// TwinCAT 3 PLC project R1_TemplatePLC
// ProgramVersion: 3.1.4022.3
// libraries:
//   Tc2_Drive, * (Beckhoff Automation GmbH)
//   Tc2_EtherCAT, * (Beckhoff Automation GmbH)
//   Tc2_IoFunctions, * (Beckhoff Automation GmbH)
//   Tc2_MC2, * (Beckhoff Automation GmbH)
//   Tc2_MC2_Drive, * (Beckhoff Automation GmbH)
//   Tc2_MDP, * (Beckhoff Automation GmbH)
//   Tc2_Standard, * (Beckhoff Automation GmbH)
//   Tc2_SUPS, * (Beckhoff Automation GmbH)
//   Tc2_System, * (Beckhoff Automation GmbH)
//   Tc2_Utilities, * (Beckhoff Automation GmbH)
//   Tc3_EventLogger, * (Beckhoff Automation GmbH)
//   Tc3_Module, * (Beckhoff Automation GmbH)
//   VisuDialogs, * (System)
// project tree:
//   DUTs/DUTsAxisOnline/FBsIO/ ST_FBGetDriveRefIO.TcDUT (not stored), ST_FBHoldingBrakeCtrlIO.TcDUT (not stored), ST_FBMotorMonitoringIO.TcDUT (not stored), ST_FBNcSWLimitSwitchCtrlIO.TcDUT (not stored), ST_FBReadChannelErrorCodeIO.TcDUT (not stored), ST_FBSetPositionOffsetIO.TcDUT, ST_McAxisOnlineErrorCollection.TcDUT, ST_McAxisStatus.TcDUT (not stored), ST_MCHaltIO.TcDUT (not stored), ST_MCHomeIO.TcDUT (not stored), ST_MCJogIO.TcDUT (not stored), ST_MCMoveAbsoluteIO.TcDUT (not stored), ST_MCMoveModuloIO.TcDUT (not stored), ST_MCMoveRelativeIO.TcDUT (not stored), ST_MCMoveVelocityIO.TcDUT (not stored), ST_MCPowerIO.TcDUT (not stored), ST_MCReadDriveAddressIO.TcDUT (not stored), ST_MCReadParameterSetIO.TcDUT (not stored), ST_MCResetIO.TcDUT (not stored), ST_MCSetPositionIO.TcDUT (not stored), ST_MCStopIO.TcDUT (not stored)
//   DUTs/DUTsAxisOnline/ ST_AX5000Diag.TcDUT (not stored), ST_McAxisOnline.TcDUT (not stored)
//   DUTs/DUTsDiagnostics/ ST_FrmWcDiag.TcDUT, ST_KBusState.TcDUT
//   DUTs/DUTsOther/ E_MachineCommand.TcDUT (not stored), E_MachineMode.TcDUT, E_MachineState.TcDUT (not stored)
//   / GlobalTextList.TcGTLO, PlcTask.TcTTO, Visualization Manager.TcVMO (not stored)
//   GVLs/ GVL.TcGVL, GVL_EventLogger_Simple.TcGVL, GVL_IO.TcGVL, GVL_Machine.TcGVL
//   GVLs/GVLsDiagnostics/ GVL_Checks.TcGVL
//   POUs/ MAIN.TcPOU, P_ErrorCollection.TcPOU, P_EventLogger_Simple.TcPOU, P_Initialization.TcPOU, P_ModeStateManager.TcPOU, P_Template.TcPOU, P_Template_SAFETY.TcPOU
//   POUs/POUsAxisOnline/AX5000/ FB_AxisDiag.TcPOU, FB_ChangeEtherCATSlaveState.TcPOU, FB_HoldingBrakeCtrlAX5000.TcPOU (not stored), FB_McAxisOnlineAX5000.TcPOU, FB_MotorMonitoringAX5000.TcPOU, FB_SetPositionOffset.TcPOU, F_AX5xErrMsg.TcPOU
//   POUs/POUsAxisOnline/AX8000/ FB_HoldingBrakeCtrlAX8000.TcPOU, FB_McAxisOnlineAX8000.TcPOU, FB_MotorMonitoringAX8000.TcPOU, FB_ReadChannelErrorCodeAX8000.TcPOU, F_AX8xErrMsg.TcPOU
//   POUs/POUsAxisOnline/EL72xx/ FB_HoldingBrakeCtrlEL72xx.TcPOU, FB_McAxisOnlineEL72xx.TcPOU, FB_MotorMonitoringEL72xx.TcPOU, FB_ReadChannelErrorCodeEL72xx.TcPOU, F_EL72ErrMsg.TcPOU
//   POUs/POUsAxisOnline/FBs/ FB_FilterEx.TcPOU (not stored), FB_GetDriveRef.TcPOU (not stored), FB_NcSWLimitSwitchCtrl.TcPOU (not stored), F_AxErrMsg.TcPOU
//   POUs/POUsAxisOnline/NC/ FB_McAxisOnlineNC.TcPOU
//   POUs/POUsDiagnostics/Checks/ CheckBounds.TcPOU, CheckDivDInt.TcPOU, CheckDivLInt.TcPOU, CheckDivLReal.TcPOU, CheckDivReal.TcPOU, CheckPointer.TcPOU, CheckRangeSigned.TcPOU, CheckRangeUnsigned.TcPOU
//   POUs/POUsDiagnostics/FB/ FB_AntiBlinkAlarmFilter.TcPOU, FB_TaskInfo.TcPOU (not stored)
//   POUs/POUsDiagnostics/ P_Checks.TcPOU, P_EtherCAT_ChangeCounter.TcPOU, P_EtherCAT_Diag.TcPOU, P_KBus.TcPOU, P_Persistent.TcPOU, P_SystemDiagnostics.TcPOU, P_SystemDiag_EventLog.TcPOU, P_SystemInfo.TcPOU, P_TaskInfo.TcPOU (not stored)
//   POUs/POUsOther/ FB_AutostartPLCHMI.TcPOU, FB_Blink_S.TcPOU
//   VISUs/VISUsAxisOnline/ PH_AxisOnline.TcVIS, PH_MotorMonitoring.TcVIS, PH_NcAxis.TcVIS
//   VISUs/ VIS_SM.TcVIS
// real-time tasks:
//   TASK PlcTask: cycle T#10ms, priority 20, ADS port 350
//   TASK SafetyTask: cycle T#10ms, priority 21, ADS port 351

CONFIGURATION R1_TemplatePLC
    RESOURCE PLC ON TwinCAT3
        TASK PlcTask(INTERVAL := T#10ms, PRIORITY := 20);
        PROGRAM MAIN WITH PlcTask : MAIN;
    END_RESOURCE
END_CONFIGURATION

// ---- DUTs/DUTsAxisOnline/FBsIO/ST_FBSetPositionOffsetIO.TcDUT
//==================================================================================================
//							Beckhoff Automation Poland
//									23.05.2018
//	Struktura zawierajaca I/O odpowiedniego bloku
//  v1.1	|| TC v 3.1.4022.16		|| - zmiana nazwy struktury usuniete CoE
//  v1.0	|| TC v 3.1.4022.16		|| - pierwsza wersja
//==================================================================================================
TYPE ST_FBSetPositionOffsetIO:
STRUCT
	bExecute						: BOOL;								// Rising edge executes cmd
	lrPosition						: LREAL;
	bRelative						: BOOL;
	eFeedback						: Tc2_MC2_Drive.E_PositionOffsetFeedback;
	eMemory							: Tc2_MC2_Drive.E_PositionOffsetMemory;
	bBusy							: BOOL;
	bError							: BOOL;
	udiErrorID						: UDINT;
	uiSecErrId						: UINT;								// Sercos Error ID for AX5000, CanOpen error ID for AX8000
END_STRUCT
END_TYPE

// ---- DUTs/DUTsAxisOnline/FBsIO/ST_McAxisOnlineErrorCollection.TcDUT
//==================================================================================================
//							Beckhoff Automation Poland
//									7.12.2018
//	Struktura zawierajaca wszsytkie bbledy AxisOnline
//  v1.1	|| TC v 3.1.4022.27		|| - dodane opisy bledow w formie zmiennych typu string
//  v1.0	|| TC v 3.1.4022.16		|| - pierwsza wersja
//==================================================================================================
TYPE ST_McAxisOnlineErrorCollection :
STRUCT
	// Error Collection
	bError							: BOOL;						// General Error flag - all error, FB, NC, drive, communication...
	bNcError						: BOOL;
	bFBError						: BOOL;						// Mc FB error
	bCommunicationError				: BOOL;						// ADS, CoE (AX8000), SoE (AX5000)...
	bDriveError						: BOOL;
	uiAdsErrorID					: UINT;						// Forwarded output FB_CoERead_ByDriveRef
	uiSecErrorID					: UINT;						// Sercos Error ID for AX5000, CanOpen error ID for AX8000
	udiErrorID						: UDINT;					// Set Position Offset FB error ID
	udiNcErrorID					: UDINT;					// Nc ErrorID
	{attribute 'displaymode':='hex'}
	udiNcErrorIDHex					: UDINT;					// Nc ErrorID
	udiFBErrorID					: UDINT;					// FB ErrorID
	{attribute 'displaymode':='hex'}
	udiFBErrorIDHex					: UDINT;					// FB ErrorID

	uiDriveErrorID					: UINT;						// 603F Error code	0x603F (Ch A)/ 0x683F (Ch B) 	UINT16
	{attribute 'displaymode':='hex'}
	uiDriveErrorIDHex				: UINT;						// 603F Error code	0x603F (Ch A)/ 0x683F (Ch B) 	UINT16
	sNcError						: STRING(255);				// Error description
	sDriveError						: STRING(255);				// Error description
END_STRUCT
END_TYPE

// ---- DUTs/DUTsDiagnostics/ST_FrmWcDiag.TcDUT
TYPE ST_FrmWcDiag :
STRUCT
	iNum					:DINT;
	sBin					:String;
END_STRUCT
END_TYPE

// ---- DUTs/DUTsDiagnostics/ST_KBusState.TcDUT
TYPE ST_KBusState :							// K_Bus_diagnostic flags structure
STRUCT
		bK_BusErr				:	BOOL;	// Bit 0 = K-Bus Err
		bTerminalStateErr		:	BOOL;	// Bit 1 = Terminal State Err
		bProcessDataLengthErr	:	BOOL;	// Bit 2 = Process Data Length Err
		bK_BusInvalid			:	BOOL;	// Bit 7 = K-Bus invalid
		bNoValidInputs			:	BOOL;	// Bit 8 = No valid Inputs
		bK_BusInputUpdateBusy	:	BOOL;	// Bit 9 = K-Bus Input Update busy
		bK_BusOutputUpdateBusy	:	BOOL;	// Bit 10 = K-Bus Output Update busy
		bWatchDogErr			:	BOOL;	// Bit 11 = Watchdog Err
		bAcycFunctionActive		:	BOOL;	// Bit 15 = Acyc. Function atcive (e.g. K-Bus Reset)
END_STRUCT
END_TYPE

// ---- DUTs/DUTsOther/E_MachineMode.TcDUT
//==================================================================================================
//							Beckhoff Automation Poland
//									22.12.2016
//	Typ glownej tablicy zdarzen historycznych
// 	v1.1	|| TC v 3.1.4022.25		|| - zamiana nazwy trybu poczatkowego na eInitialization
// 	v1.0	|| TC v 3.1.4020.28		|| - pierwsza wersja
//==================================================================================================
{attribute 'strict'}
{attribute 'qualified_only'}
TYPE E_MachineMode :
(
	eInitialization			:= 0,
	eManual					:= 1,
	eMaintenance			:= 2,
	eAutomatic				:= 3,
	eSemiAutomatic			:= 4,
	eFirstFilling			:= 5,
	eEmptying				:= 6
);
END_TYPE

// ---- GVLs/GVL.TcGVL
{attribute 'qualified_only'}
VAR_GLOBAL CONSTANT
	byNoOfAxes 							: BYTE:= 10; 			// Liczba osi
END_VAR
VAR_GLOBAL
	Axis								: ARRAY [1..byNoOfAxes] OF AXIS_REF;
	stMcAxisOnline						: ARRAY [1..byNoOfAxes] OF ST_McAxisOnline;
	//
	bAllUnitsReady						: BOOL;					// All machine units are OK, and ready to operate
	bGeneralOK							: BOOL;					// There is no Warning, Error or Fatal Error - just when it's true - You can operate
	bGeneralWarning						: BOOL;					// Warning - just message/event - no reaction
	bGeneralError						: BOOL;					// Error - machine has to stop, start is possible from this position
	bGeneralFatalError					: BOOL;					// Fatal error causes machine stop. You have to go back for cycle begin.

	// 
	bRestartRequired					: BOOL;					// In case of fatal error, when whole process restart required
	bMuteGeneralError					: BOOL;					// Just for service/maitenance - if You are aware of consequences You can force muting mode
	bMuteGeneralFatalError				: BOOL;					// Just for service/maitenance - if You are aware of consequences You can force muting mode
END_VAR

// ---- GVLs/GVLsDiagnostics/GVL_Checks.TcGVL
{attribute 'qualified_only'}
VAR_GLOBAL PERSISTENT
	dCheckBounds					: DINT;			// Licznik przekroczen zakresu indexow, np. tablic
	dCheckDivDInt					: DINT;			// Licznik prob dzielenia Dint przez 0
	dCheckDivLInt					: DINT; 		// Licznik prob dzielenia LInt przez 0
	dCheckDivLReal					: DINT; 		// Licznik prob dzielenia LREAL przez 0
	dCheckDivReal					: DINT; 		// Licznik prob dzielenia REAL przez 0
	dCheckRangeSigned				: DINT;			// Licznik przekroczen liczby znakowej
	dCheckRangeUnsigned				: DINT; 		// Licznik przekroczen liczby bezznakowej
END_VAR

// ---- GVLs/GVL_EventLogger_Simple.TcGVL
{attribute 'qualified_only'}
VAR_GLOBAL
	arrMessageTriggers		: ARRAY [1..nMaxNumMessages] OF BOOL; // auto clear
	arrWarningTriggers		: ARRAY [1..nMaxNumWarnings] OF BOOL; // auto clear
	arrErrorTriggers 		: ARRAY [1..nMaxNumErrors] OF BOOL; // manual clear
	arrErrorConfirmations	: ARRAY [1..nMaxNumErrors] OF BOOL; // auto clear
END_VAR
VAR_GLOBAL CONSTANT
	nMaxNumMessages 	: UDINT := 3;
	nMaxNumWarnings 	: UDINT := 3;
	nMaxNumErrors 		: UDINT := 3;
END_VAR

// ---- GVLs/GVL_IO.TcGVL
{attribute 'qualified_only'}
VAR_GLOBAL
// =============== SAMPLE NAMES =================

	di_PBStart 					AT %I*	: BOOL;					// Push button - Start
	di_PBStop 					AT %I*	: BOOL;					// Push button - Stop
	di_PBReset 					AT %I*	: BOOL;					// Push button - Reset
// ==============================================
// =================== SAFETY ===================
	bSAFETY_Error				AT %I*	: BOOL;
	bSAFETY_ResetCMD 			AT %Q*	: BOOL;
	bSAFETY_ResetBusy			AT %I*	: BOOL;
	bSAFETY_PermissionSS1		AT %I*	: BOOL; 				// Sygnal NC - TRUE - pozwolenie na prace
	bSAFETY_PermissionSS2		AT %I*	: BOOL; 				// Sygnal NC - TRUE - pozwolenie na prace
// ======== Error and states collection =========
	dwGroupErrors				AT %I*	: DWORD;				// Group Error collection - Communication, FB, Other...
	dwAXStatesSTO				AT %I*	: DWORD;
	dwAXStatesSOS				AT %I*	: DWORD;
	dwAXErrors					AT %I*	: DWORD;
END_VAR

// ---- GVLs/GVL_Machine.TcGVL
{attribute 'qualified_only'}
VAR_GLOBAL
	eMode									: E_MachineMode := E_MachineMode.eInitialization;	// Global machine mode
																						(*	eInitialization			:= 0,
																							eManual					:= 1,
																							eMaintenance			:= 2,
																							eAutomatic				:= 3,
																							eSemiAutomatic			:= 4,
																							eFirstFilling			:= 5,
																							eEmptying				:= 6	*)
																							
	eCommand								: E_MachineCommand; 							// Global machine command
																						(*	eAbort	  				:= 10,
																							eStop	  				:= 20,
																							eRun 	  				:= 30,
																							eReset	  				:= 40	*)
																							
	eState									: E_MachineState; 								// Global machine state
																						(*	eIdle					:= 0,
																							eAborting				:= 10,
																							eAborted				:= 20,
																							eStopping				:= 30,
																							eStopped				:= 40,
																							eStarting				:= 50,
																							eRunning				:= 60,
																							eReseting				:= 70,
																							eError					:= 1000	*)
END_VAR

// ---- POUs/MAIN.TcPOU
//==================================================================================================
//							Beckhoff Automation Poland
//									02.11.2018
//	Projekt startowy
// 	v1.2	|| TC v 3.1.4022.4		|| - zmiana wywolania osi
// 	v1.1	|| TC v 3.1.4020.32		|| - Aktualizacja
// 	v1.0	|| TC v 3.1.4020.28		|| - Pierwsza wersja
//==================================================================================================
PROGRAM MAIN
VAR
END_VAR

P_SystemDiagnostics();

P_EventLogger_Simple();

P_ErrorCollection();

P_ModeStateManager();

P_Template_SAFETY(eMachineMode:= GVL_Machine.eMode, eMachineCommand:= GVL_Machine.eCommand, eMachineState=> , bError=> );

P_Template(eMachineMode:= GVL_Machine.eMode, eMachineCommand:= GVL_Machine.eCommand, eMachineState=> , Axis1 := GVL.Axis[1]);
(*
P_Template_CAM(	eMachineMode		:= GVL_Machine.eMode, 
				eMachineCommand		:= GVL_Machine.eCommand, 
				eMachineState		=> GVL_Machine.eState,
				Axis1				:= GVL.Axis[1], 
				Axis2				:= GVL.Axis[2], 
				Axis3				:= GVL.Axis[3]);
*)

END_PROGRAM

// ---- POUs/POUsDiagnostics/P_SystemDiagnostics.TcPOU
//==================================================================================================
//							Beckhoff Automation Poland
//									2.11.2018
//					Program zbiorczy diagnostyki systemu
// 
//	v1.4 	|| TC v 3.1.4022.25 	|| Dodany state machine
//	v1.3 	|| TC v 3.1.4022.20 	|| Usuniete P_MDP, dodany podprogram EventLoggera P_SystemDiag_EventLog
//	v1.2 	|| TC v 3.1.4020.32 	|| Dodane P_EtherCAT_ChangeCounter
//	v1.1 	|| TC v 3.1.4020.14 	|| Dodane wyjscia bOk, bWarning, bError
//	v1.0 	|| TC v 3.1.4020.0 		|| Pierwsza wersja
//==================================================================================================
PROGRAM P_SystemDiagnostics
VAR_INPUT
	eMachineMode							: E_MachineMode; 		// Machine mode
	eMachineCommand							: E_MachineCommand; 	// Command from top level state program
END_VAR
VAR_OUTPUT
	eMachineState							: E_MachineState;
	bOK										: BOOL;					// Brak bledow i ostrzezen
	bWarning								: BOOL;					// Ostrzezenie
	bError									: BOOL;					// Zbiorcza flaga bledow
END_VAR
VAR
END_VAR

P_SystemInfo(bConfirm:=);
P_Persistent();
P_EtherCAT_Diag();
P_EtherCAT_ChangeCounter(bReset := );
P_KBus();
P_Checks(bReset := );
P_TaskInfo();

// Machine mode change over
CASE eMachineMode OF
	
	E_MachineMode.eInitialization:
		; // Do nothing
	
ELSE
	
	// Set flags
	bError										:= P_SystemInfo.bError OR P_Persistent.bError OR P_EtherCAT_Diag.bError OR P_EtherCAT_ChangeCounter.bError OR P_KBus.bError OR P_Checks.bError OR P_TaskInfo.bError;
	bWarning									:= P_SystemInfo.bWarning OR P_Persistent.bWarning OR P_EtherCAT_Diag.bWarning OR P_EtherCAT_ChangeCounter.bWarning OR P_KBus.bWarning OR P_Checks.bWarning OR P_TaskInfo.bWarning;
	bOk											:= NOT (bError OR bWarning);
	
	// State machine
	CASE eMachineState OF
	
		E_MachineState.eIdle, E_MachineState.eStopping, E_MachineState.eStopped, E_MachineState.eStarting, E_MachineState.eAborting, E_MachineState.eAborted:

			// Ignore global commands eAbort, eRun, eStop, eReset, eRestart
			// Set eRunning state
			eMachineState 						:= E_MachineState.eRunning;

		E_MachineState.eRunning:
		
			// Ignore global commands eAbort, eRun, eStop, eReset, eRestart
			// If error go to error state
			IF bError THEN
				eMachineState					:= E_MachineState.eError;
			END_IF
	
		E_MachineState.eRestarting, E_MachineState.eReseting:

			// Reset/Restart only if not OK
			P_EtherCAT_ChangeCounter.bReset		:= NOT P_EtherCAT_ChangeCounter.bOK;
			P_Checks.bReset						:= NOT P_Checks.bOK;
			IF NOT bError THEN
				eMachineState					:= E_MachineState.eRunning;
			END_IF

		E_MachineState.eError:
	
			IF eMachineCommand = E_MachineCommand.eReset THEN
				eMachineState					:= E_MachineState.eReseting;
			END_IF
	
			IF eMachineCommand = E_MachineCommand.eRestart THEN
				eMachineState					:= E_MachineState.eRestarting;
			END_IF
	
	END_CASE
	
END_CASE

// Log to events - You can switch it off in Initialization phase
P_SystemDiag_EventLog();

END_PROGRAM

// ---- POUs/POUsDiagnostics/P_SystemInfo.TcPOU
//==================================================================================================
//							Beckhoff Automation Poland
//									P_SystemInfo
//									31.10.2018
//					Program odczytujący informacje o TC Runtime
// 
//	v1.2 	|| TC v 3.1.4022.25 	|| - bOK dodane BSOD i sprawdzenie licencji
//	v1.1 	|| TC v 3.1.4020.14 	|| - Dodane wyjscia bOk, bWarning, bError
//	v1.0 	|| TC v 3.1.4020.0 		|| - Pierwsza wersja
//==================================================================================================
PROGRAM P_SystemInfo
VAR_INPUT
	bConfirm					: BOOL;					// Potwierdzenie bledu/ostrzezenia persistentow - blad/ostrzezenie nie znika, my usuwamy flage error lub warning
END_VAR
VAR_OUTPUT
	bOK							: BOOL;					// Zmienne wczytane prawidlowo
	bWarning					: BOOL;					// Zmienne wczytane z pliku zapasowego
	bError						: BOOL;					// Nie wczytano zmiennych
END_VAR
VAR
	sStartTime					: STRING;				// Przekonwertowany czas
END_VAR

//_AppInfo.ObjId; 			(* Object ID of the PLC project instance *)
//_AppInfo.TaskCnt;			(* The number of tasks in the actual runtime system *)
//_AppInfo.OnlineChangeCnt;	(* The number of online changes made since the last complete download. *)
//_AppInfo.Flags;				(* Reserved for future use *)
//_AppInfo.AdsPort; 			(* ADS port of PLC application *)
bOK							:= (_AppInfo.BootDataLoaded OR bConfirm) AND NOT _AppInfo.LicensesPending AND NOT _AppInfo.BSODOccured;	(* PERSISTENT variables: LOADED (without error) *)
bWarning					:= _AppInfo.OldBootData AND NOT bConfirm;	(* PERSISTENT variables: INVALID (the back-up copy was loaded, since no valid data was present) *)
bError						:= NOT bOK AND NOT bWarning;
//_AppInfo.KeepOutputsOnBP;	(* The flag can be set to avoid that the outputs are zero-filled if a breakpoint is reached. The task keeps running. Only the execution of PLC code is interrupted. *)
//_AppInfo.TComSrvPtr;		(* Pointer to TcCOM Object Server *)
//_AppInfo.AppName;			(* TwinCAT generated name containing the port number. *)
//_AppInfo.ProjectName;		(* The name of the PLC project. *)
sStartTime					:= DELETE(DT_TO_STRING(_AppInfo.AppTimestamp),3,1);(* Date and time of application start *)
(*_AppInfo.BSODOccured;
_AppInfo.LicensesPending;
_AppInfo.ShutdownInProgress;*)

END_PROGRAM

// ---- POUs/POUsDiagnostics/P_Persistent.TcPOU
//==================================================================================================
//							Beckhoff Automation Poland
//									25.04.2018
//		Program obslugujacy pamiec nieulotna 
// 	v1.3	|| TC v 3.1.4022.16		|| - Przeniesienie logowania do EvenLogger'a do programu P_SystemDiag_EventLog
// 	v1.2	|| TC v 3.1.4022.0		|| - Dodanie akcji UPS
//	v1.1 	|| TC v 3.1.4020.14 	|| - Dodane wyjscia bOk, bWarning, bError
//	v1.0 	|| TC v 3.1.4020.0 		|| - Pierwsza wersja
//==================================================================================================
PROGRAM P_Persistent
VAR_INPUT
	bWrite						: BOOL;						// Zapis na rozkaz - tylko dla iType = 0 lub nieokreslonego, gdy używany jest FB_WritePersistentData
	tInterval					: TIME := T#1H;				// Czestotliwosc zapisu na karte CF - tylko dla iType = 0 lub nieokreslonego, gdy używany jest FB_WritePersistentData
END_VAR
VAR_OUTPUT
	// Brak obslugi
	bOK							: BOOL := TRUE;				// Brak bledow i ostrzezen
	bWarning					: BOOL;						// Ostrzezenie
	bError						: BOOL;						// Zbiorcza flaga bledow
END_VAR
VAR
	iType						: INT := 0;					(* typ zapisu persistent:
																0: standardowo - na zadanie oraz co okreslony czas
																10: FB_S_UPS, np: CX50x0,C6915-0000,CP62xx-0020,CP77xx-0030
																20: FB_S_UPS_CB3011, np: CP66xx-0020, CP26xx-0000
																30: FB_S_UPS_CX51x0, np: CX51x0
																40: FB_S_UPS_CX9020_U900, np: CX9020 *)
	fbS_UPS						: FB_S_UPS;
	fbS_UPS_CB3011				: FB_S_UPS_CB3011;
	fbS_UPS_CX51x0				: FB_S_UPS_CX51x0;
	fbS_UPS_CX9020_U900			: FB_S_UPS_CX9020_U900;
	fbS_UPS_BAPI				: FB_S_UPS_BAPI;
	// Obsługa ogólna
	fbWritePersistentData 		: FB_WritePersistentData;	// Blok zapisu
	T1							: TON;						// Timer zapisu
END_VAR

CASE iType OF
	0:
		A_WritePersistentData();
		
	10:
	
		A_fbS_UPS();
		
	20:
		
		A_fbS_UPS_CB3011();
		
	30:
	
		A_fbS_UPS_CX51x0();
		
	40:
	
		A_fbS_UPS_CX9020_U900();
		
	50:
	
		A_fbS_UPS_BAPI();
		
ELSE
		A_WritePersistentData();		
		
END_CASE

ACTION A_fbS_UPS:
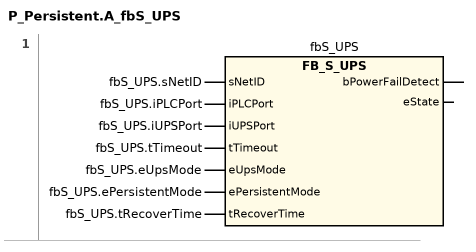
// NETWORK 1
fbS_UPS(
    sNetID := fbS_UPS.sNetID,
    iPLCPort := fbS_UPS.iPLCPort,
    iUPSPort := fbS_UPS.iUPSPort,
    tTimeout := fbS_UPS.tTimeout,
    eUpsMode := fbS_UPS.eUpsMode,
    ePersistentMode := fbS_UPS.ePersistentMode,
    tRecoverTime := fbS_UPS.tRecoverTime); // FB_S_UPS
END_ACTION

ACTION A_fbS_UPS_BAPI:
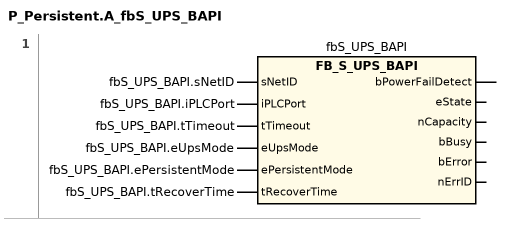
// NETWORK 1
fbS_UPS_BAPI(
    sNetID := fbS_UPS_BAPI.sNetID,
    iPLCPort := fbS_UPS_BAPI.iPLCPort,
    tTimeout := fbS_UPS_BAPI.tTimeout,
    eUpsMode := fbS_UPS_BAPI.eUpsMode,
    ePersistentMode := fbS_UPS_BAPI.ePersistentMode,
    tRecoverTime := fbS_UPS_BAPI.tRecoverTime); // FB_S_UPS_BAPI
END_ACTION

ACTION A_fbS_UPS_CB3011:
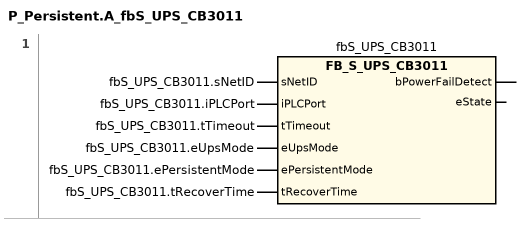
// NETWORK 1
fbS_UPS_CB3011(
    sNetID := fbS_UPS_CB3011.sNetID,
    iPLCPort := fbS_UPS_CB3011.iPLCPort,
    tTimeout := fbS_UPS_CB3011.tTimeout,
    eUpsMode := fbS_UPS_CB3011.eUpsMode,
    ePersistentMode := fbS_UPS_CB3011.ePersistentMode,
    tRecoverTime := fbS_UPS_CB3011.tRecoverTime); // FB_S_UPS_CB3011
END_ACTION

ACTION A_fbS_UPS_CX51x0:
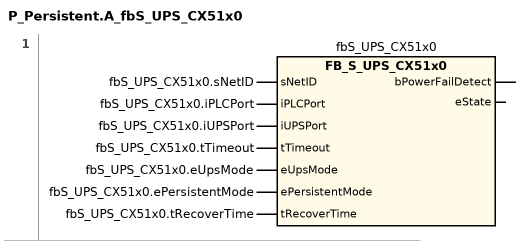
// NETWORK 1
fbS_UPS_CX51x0(
    sNetID := fbS_UPS_CX51x0.sNetID,
    iPLCPort := fbS_UPS_CX51x0.iPLCPort,
    iUPSPort := fbS_UPS_CX51x0.iUPSPort,
    tTimeout := fbS_UPS_CX51x0.tTimeout,
    eUpsMode := fbS_UPS_CX51x0.eUpsMode,
    ePersistentMode := fbS_UPS_CX51x0.ePersistentMode,
    tRecoverTime := fbS_UPS_CX51x0.tRecoverTime); // FB_S_UPS_CX51x0
END_ACTION

ACTION A_fbS_UPS_CX9020_U900:
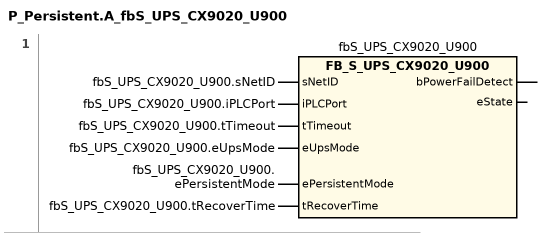
// NETWORK 1
fbS_UPS_CX9020_U900(
    sNetID := fbS_UPS_CX9020_U900.sNetID,
    iPLCPort := fbS_UPS_CX9020_U900.iPLCPort,
    tTimeout := fbS_UPS_CX9020_U900.tTimeout,
    eUpsMode := fbS_UPS_CX9020_U900.eUpsMode,
    ePersistentMode := fbS_UPS_CX9020_U900.ePersistentMode,
    tRecoverTime := fbS_UPS_CX9020_U900.tRecoverTime); // FB_S_UPS_CX9020_U900
END_ACTION

ACTION A_WritePersistentData:
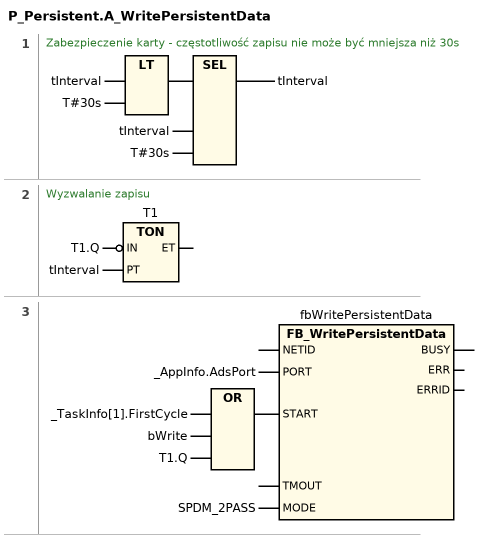
// NETWORK 1
// Zabezpieczenie karty - częstotliwość zapisu nie może być mniejsza niż 30s
tInterval := SEL(tInterval < T#30s, tInterval, T#30s);

// NETWORK 2
// Wyzwalanie zapisu
T1(IN := NOT T1.Q, PT := tInterval); // TON

// NETWORK 3
fbWritePersistentData(
    PORT := _AppInfo.AdsPort,
    START := _TaskInfo[1].FirstCycle OR bWrite OR T1.Q,
    MODE := SPDM_2PASS); // FB_WritePersistentData
END_ACTION

END_PROGRAM

// ---- POUs/POUsDiagnostics/P_EtherCAT_Diag.TcPOU
//==================================================================================================
//							Beckhoff Automation Poland
//									18.06.2018
//		Program wysyłający błędy magistrali EBus do EvenLogger'a
//
//	v1.4	|| TC v 3.1.4022.16		|| - Przeniesiono logowanie do EventLoggera wraz z zabepieczeniem przed zbyt szybkim logowaniem zdarzeń do programu P_SystemDiag_EventLog. 
//	v1.3	|| TC v 3.1.4020.28		|| - Dodano zabezpieczenie przed zbyt sczęstym logowaniem eventów i zmieniono system logowania błędów ramek. Od teraz każda ramka ma swój EventId. Wstępnie zarezerwowano 8 ramek.
//  v1.2	|| TC v 3.1.4020.28		|| - Usunięto zbędne wejścia (sFormat, pDataAdr i udiDataLen) na fbDevDiag które podoowały generowanie błędów przekroczeń indeksów
//									|| - Dodano logowanie do EventLoggera 
//	v1.1 	|| TC v 3.1.4020.14 	|| - Dodane wyjscia bOk, bWarning, bError
//	v1.0 	|| TC v 3.1.4020.0 		|| - Pierwsza wersja
//==================================================================================================
PROGRAM P_EtherCAT_Diag
VAR CONSTANT
	iNumOfFrames				: INT := 8;							// Liczba FrmWcState
END_VAR
VAR_OUTPUT
	bOK							: BOOL;								// Brak bledow i ostrzezen
	bWarning					: BOOL;								// Ostrzezenie - nie wystepuja w tym podprogramie - wystepuja dla zachowania spojnosci
	bError						: BOOL;								// Zbiorcza flaga bledow
END_VAR
VAR
	uiDevState		AT %I*		: UINT;								// DevState mastera EtherCAT'a
																	(*	0x0001 = Link error
																		0x0002 = I/O locked after link error (I/O reset required)
																		0x0004 = Link error (redundancy adapter)
																		0x0008 = Missing one frame (redundancy mode)
																		0x0010 = Out of send resources (I/O reset required)
																		0x0020 = Watchdog triggered
																		0x0040 = Ethernet driver (miniport) not found
																		0x0080 = I/O reset active
																		0x0100 = At least one device in 'INIT' state
																		0x0200 = At least one device in 'PRE-OP' state
																		0x0400 = At least one device in 'SAFE-OP' state
																		0x0800 = At least one device indicates an error state
																		0x1000 = DC not in sync*)
	uiFrmWcState		AT %I*	: ARRAY[1..iNumOfFrames] OF UINT;	// FrmWcState
																	(*	0x0001 = wrong working counter of 1. EtherCAT command received
																		0x0002 = wrong working counter of 2. EtherCAT command received
																		0x0004 = wrong working counter of 3. EtherCAT command received
																		...
																		...
																		0x4000 = wrong working counter of 15. EtherCAT command received
																		0x8000 = complete frame missing*)
	iIterator					: INT;
END_VAR

bError 									:= uiDevState <> 0;							// Ustawienie flagi bledu zgodnie z uiDevState

FOR iIterator := 1 TO iNumOfFrames DO
	IF uiFrmWcState[iIterator] <> 0 THEN
		bError 							:= TRUE;									// Ustawienei flagi bledu gdy chociaz jeden frame jest z bledem
		EXIT;
	END_IF
END_FOR

bOK 									:= NOT bError AND NOT bWarning;

END_PROGRAM

// ---- POUs/POUsDiagnostics/P_EtherCAT_ChangeCounter.TcPOU
//==================================================================================================
//							Beckhoff Automation Poland
//									19.10.2018
// Program wyświetlający informację o licznikach State Changes i NOT Present - opis ponizej
// Wymagane jest podanie jedynie adresu AMS NET ID Mastera EtherCATa i liczby urzadzen Slave
// State Changes/Not Present
// State Changes - for example if the sync task needs longer then 100ms, state changes from OP to other, but Slave is present
// Not Present - If it switchs back from OP (power off, broken...)
//
//	v1.3 	|| TC v 3.1.4022.25		 	|| - Reset as an input, Presen --> Present 
//	v1.2 	|| TC v 3.1.4022.20		 	|| - Return instruction and some comments
//	v1.1 	|| TC v 3.1.4020.32		 	|| - Dodane wyjscia bOk, bWarning, bError, opisu, zmiana typow zmiennych
//	v1.0 	|| TC v 3.1.4020.32 		|| - Pierwsza wersja
//==================================================================================================
PROGRAM P_EtherCAT_ChangeCounter
VAR CONSTANT
	sAmsNetID_EtherCATMaster				: T_AmsNetId	:= '';							// EtherCAT Master AMS Net ID
	wCountOfEtherCATSlaves					: WORD 			:= 10; 							// Count of EtherCAT Slaves
END_VAR
VAR_INPUT
	bReset									: BOOL;
END_VAR
VAR_OUTPUT
	bOK										: BOOL;											// Brak bledow i ostrzezen
	bWarning								: BOOL;											// Ostrzezenie - nie wystepuja w tym podprogramie - wystepuja dla zachowania spojnosci
	bError									: BOOL;											// Zbiorcza flaga bledow
END_VAR
VAR
	//======================= State Changes/ ========================
	arrAbnormalStateChangeCounter			: ARRAY [1..wCountOfEtherCATSlaves] OF DWORD; 	// State Changes/  - tablica zawieraca dane dla poszczegilnych Slave
	wAbnormalStateChangeCounterPosition		: WORD;											// Pozycja pierwszego Slavea który zmienił wartosc licznika
	bAbnormalStateChangeCounterChanged		: BOOL;											// Flaga wystapienia zmiany licznika
	//===============================================================
	//======================== /Not Present =========================
	arrPresentStateChangeCounter			: ARRAY [1..wCountOfEtherCATSlaves] OF DWORD; 	// /Not Present  - tablica zawieraca dane dla poszczegilnych Slave
	wPresentStateChangeCounterPosition		: WORD;											// Pozycja pierwszego Slavea który zmienił wartosc licznika
	bPresentStateChangeCounterChanged		: BOOL;											// Flaga wystapienia zmiany licznika
	//===============================================================
	//======================= Internal ==============================
	bFirstCycle								: BOOL := TRUE;
	tonRefresh								: TON;
	tRefreshTime							: TIME := T#200MS;								// Refresh timer
	
	//===============================================================
	//=================== Internal hidden ===========================
	{attribute 'hide'}
	fbADSREAD_AbnormalStateChangeCounter	: ADSREAD;
	{attribute 'hide'}
	fbADSREAD_PresentStateChangeCounter		: ADSREAD;
	{attribute 'hide'}
	arrAbnormalStateChangeCounterOld		: ARRAY [1..wCountOfEtherCATSlaves] OF DWORD; 	// Stara tablica - do celow porownawczych
	{attribute 'hide'}
	arrPresenStateChangeCounterOld			: ARRAY [1..wCountOfEtherCATSlaves] OF DWORD; 	// Stara tablica - do celow porownawczych
	{attribute 'hide'}
	i										: WORD;
	{attribute 'hide'}
	ft1										: F_TRIG;
	{attribute 'hide'}
	ft2										: F_TRIG;
	//===============================================================
END_VAR

{region "Is it ready to read?"}
IF sAmsNetID_EtherCATMaster = '' OR wCountOfEtherCATSlaves = 0 THEN
	RETURN;
END_IF
{endregion}
{region "Call FBs"}
// Start reading
tonRefresh(IN:= NOT tonRefresh.Q, PT:= tRefreshTime);

// End of reading 
ft1(CLK:= fbADSREAD_PresentStateChangeCounter.BUSY);
ft2(CLK:= fbADSREAD_AbnormalStateChangeCounter.BUSY);

// Reading
fbADSREAD_PresentStateChangeCounter(
	NETID			:= sAmsNetID_EtherCATMaster,
	PORT			:= 16#FFFF,
	IDXGRP			:= 16#16,
	IDXOFFS			:= 0,
	LEN				:= SIZEOF(arrPresentStateChangeCounter),
	DESTADDR		:= ADR(arrPresentStateChangeCounter),
	READ			:= tonRefresh.Q);

fbADSREAD_AbnormalStateChangeCounter(
	NETID			:= sAmsNetID_EtherCATMaster,
	PORT			:= 16#FFFF,
	IDXGRP			:= 16#13,
	IDXOFFS			:= 0,
	LEN				:= SIZEOF(arrAbnormalStateChangeCounter),
	DESTADDR		:= ADR(arrAbnormalStateChangeCounter),
	READ			:= ft1.Q);
{endregion}
{region "Change detection"}
//================= Checks positon of change ====================
// Check if changed
IF ft1.Q THEN
	IF NOT  bFirstCycle THEN
		FOR i := 1 TO wCountOfEtherCATSlaves DO
			IF arrPresentStateChangeCounter[i] <> arrPresenStateChangeCounterOld[i] THEN
				wPresentStateChangeCounterPosition 		:= i;
				bPresentStateChangeCounterChanged 		:= TRUE;
				EXIT;
			END_IF
		END_FOR
	END_IF
	arrAbnormalStateChangeCounterOld 					:= arrAbnormalStateChangeCounter;
END_IF

IF ft2.Q THEN
	IF NOT  bFirstCycle THEN
		FOR i := 1 TO wCountOfEtherCATSlaves DO
			IF arrAbnormalStateChangeCounter[i] <> arrAbnormalStateChangeCounterOld[i] THEN
				wAbnormalStateChangeCounterPosition 	:= i;
				bAbnormalStateChangeCounterChanged 		:= TRUE;
				EXIT;
			END_IF
		END_FOR
	END_IF
	arrPresenStateChangeCounterOld 						:= arrPresentStateChangeCounter;
	bFirstCycle 										:= FALSE;
END_IF
//===============================================================
{endregion}
{region "Reset and states"}
//  Reset
IF bReset THEN
	wPresentStateChangeCounterPosition 					:= 0;
	wAbnormalStateChangeCounterPosition 				:= 0;
	bPresentStateChangeCounterChanged 					:= FALSE;
	bAbnormalStateChangeCounterChanged 					:= FALSE;
	bReset 												:= FALSE;
END_IF

// Set outputs
bError 			:= bPresentStateChangeCounterChanged OR bAbnormalStateChangeCounterChanged;
bOK 			:= NOT bError AND NOT bWarning;
{endregion}

END_PROGRAM

// ---- POUs/POUsDiagnostics/P_KBus.TcPOU
//==================================================================================================
//							Beckhoff Automation Poland
//									P_KBus
//								15.06.2018
//					Program wysyłający błędy magistrali KBus do EvenLogger'a
// 
//	v1.3	|| TC v 3.1.4022.20		|| - Przeniesiono logowanie do EventLoggera wraz z zabepieczeniem przed zbyt szybkim logowaniem zdarzeń do programu P_SystemDiag_EventLog. 
//	v1.2	|| TC v 3.1.4020.28		|| - Dodano zabezpieczenie przed zbyt częstym logowaniem eventów
//	v1.1 	|| TC v 3.1.4020.14 	|| - Dodane wyjscia bOk, bWarning, bError
//	v1.0 	|| TC v 3.1.4020.0 		|| - Pierwsza wersja
//==================================================================================================
PROGRAM P_KBus
VAR_OUTPUT
	// Brak obslugi
	bOK								: BOOL := TRUE;			// Brak bledow i ostrzezen
	bWarning						: BOOL;					// Ostrzezenie
	bError							: BOOL;					// Zbiorcza flaga bledow
END_VAR
VAR
	uiKbusState	AT %I*				: UINT;		// K-Bus Box State << PLEASE LINK THIS VARIABLE WITH YOUR BOX (Devices > Device > Box > Inputs > State)
	stKBusState						: ST_KBusState;	// K_Bus_diagnostic errors structure
END_VAR

// Read Error flags form K-Bus Device
stKBusState.bK_BusErr				:=	uiKbusState.0;		// Bit 0 = K-Bus Err
stKBusState.bTerminalStateErr		:=	uiKbusState.1;		// Bit 1 = Terminal State Err
stKBusState.bProcessDataLengthErr	:=	uiKbusState.2;		// Bit 2 = Process Data Length Err
stKBusState.bK_BusInvalid			:=	uiKbusState.7;		// Bit 7 = K-Bus invalid
stKBusState.bNoValidInputs			:=	uiKbusState.8;		// Bit 8 = No valid Inputs
stKBusState.bK_BusInputUpdateBusy	:=	uiKbusState.9;		// Bit 9 = K-Bus Input Update busy	
stKBusState.bK_BusOutputUpdateBusy	:=	uiKbusState.10;		// Bit 10 = K-Bus Output Update busy
stKBusState.bWatchDogErr			:=	uiKbusState.11;		// Bit 11 = Watchdog Err
stKBusState.bAcycFunctionActive		:=	uiKbusState.15;		// Bit 15 = Acyc. Function atcive (e.g. K-Bus Reset)

END_PROGRAM

// ---- POUs/POUsDiagnostics/P_Checks.TcPOU
//==================================================================================================
//							Beckhoff Automation Poland
//									19.10.2018
//	Program wykrywajacy bledy dzielnia przez 0 i przekraczania zakresow zmiennych, tablic...
// 
//	v1.4	|| TC v 3.1.4022.25		|| - Ustawiono setowanie bledow, dodano wejscie bReset 
//	v1.3	|| TC v 3.1.4022.16		|| - Przeniesiono logowanie do EventLoggera wraz z zabepieczeniem przed zbyt szybkim logowaniem zdarzeń do programu P_SystemDiag_EventLog. 
//	v1.2	|| TC v 3.1.4020.28		|| - Dodano logowanie do EventLoggera wraz z zabepieczeniem przed zbyt szybki logowaniem zdarzeń
//	v1.1 	|| TC v 3.1.4020.14 	|| - Dodane wyjscia bOk, bWarning, bError
//	v1.0 	|| TC v 3.1.4020.0 		|| - Pierwsza wersja
//==================================================================================================
PROGRAM P_Checks
VAR_INPUT
	bReset							: BOOL;
END_VAR
VAR_OUTPUT
	bOK								: BOOL;	// Brak bledow i ostrzezen
	bWarning						: BOOL;	// Ostrzezenie - nie wystepuja w tym podprogramie - wystepuja dla zachowania spojnosci
	bError							: BOOL;	// Zbiorcza flaga bledow
END_VAR
VAR
	bCheckBounds					: BOOL;	// Flaga przekroczen zakresu indexow, np. tablic
	bCheckDivDInt					: BOOL;	// Flaga prob dzielenia Dint przez 0
	bCheckDivLInt					: BOOL; // Flaga prob dzielenia LInt przez 0
	bCheckDivLReal					: BOOL; // Flaga prob dzielenia LREAL przez 0
	bCheckDivReal					: BOOL; // Flaga prob dzielenia REAL przez 0
	bCheckRangeSigned				: BOOL;	// Flaga przekroczen liczby znakowej
	bCheckRangeUnsigned				: BOOL; // Flaga przekroczen liczby bezznakowej
	
	dCheckBoundsOld					: DINT;	// Licznik przekroczen zakresu indexow, np. tablic
	dCheckDivDIntOld				: DINT;	// Licznik prob dzielenia Dint przez 0
	dCheckDivLIntOld				: DINT; // Licznik prob dzielenia LInt przez 0
	dCheckDivLRealOld				: DINT; // Licznik prob dzielenia LREAL przez 0
	dCheckDivRealOld				: DINT; // Licznik prob dzielenia REAL przez 0
	dCheckRangeSignedOld			: DINT;	// Licznik przekroczen  liczby znakowej
	dCheckRangeUnsignedOld			: DINT; // Licznik przekroczen  liczby bezznakowej
END_VAR

IF bReset THEN
	bCheckBounds 					:= FALSE;
	bCheckDivDInt					:= FALSE;
	bCheckDivLInt					:= FALSE;
	bCheckDivLReal					:= FALSE;
	bCheckDivReal					:= FALSE;
	bCheckRangeSigned				:= FALSE;
	bCheckRangeUnsigned				:= FALSE;
ELSE
	bCheckBounds 					S= dCheckBoundsOld <> GVL_Checks.dCheckBounds;
	bCheckDivDInt					S= dCheckDivDIntOld <> GVL_Checks.dCheckDivDInt;
	bCheckDivLInt					S= dCheckDivLIntOld <> GVL_Checks.dCheckDivLInt;
	bCheckDivLReal					S= dCheckDivLRealOld <> GVL_Checks.dCheckDivLReal;
	bCheckDivReal					S= dCheckDivRealOld <> GVL_Checks.dCheckDivReal;
	bCheckRangeSigned				S= dCheckRangeSignedOld <> GVL_Checks.dCheckRangeSigned;
	bCheckRangeUnsigned				S= dCheckRangeUnsignedOld <> GVL_Checks.dCheckRangeUnsigned;	
END_IF

dCheckBoundsOld 					:= GVL_Checks.dCheckBounds;
dCheckDivDIntOld 					:= GVL_Checks.dCheckDivDInt;
dCheckDivLIntOld 					:= GVL_Checks.dCheckDivLInt;
dCheckDivLRealOld 					:= GVL_Checks.dCheckDivLReal;
dCheckDivRealOld 					:= GVL_Checks.dCheckDivReal;
dCheckRangeSignedOld 				:= GVL_Checks.dCheckRangeSigned;
dCheckRangeUnsignedOld 				:= GVL_Checks.dCheckRangeUnsigned;

bError 								:= bCheckBounds OR bCheckDivDInt OR bCheckDivLInt OR bCheckDivLReal OR bCheckDivReal OR bCheckRangeSigned OR bCheckRangeUnsigned;
bOK 								:= NOT bError AND NOT bWarning;

END_PROGRAM

// ---- POUs/POUsDiagnostics/P_SystemDiag_EventLog.TcPOU
//==================================================================================================
//							Beckhoff Automation Poland
//									29.09.2020
//	Program logowanie do EventLoggera wraz z zabepieczeniem przed zbyt szybkim logowaniem zdarzen
//	Dziala tylko w polaczeniu z podprogramami i z blokami FB_AdvancedLogEvent, FB_AntiBlinkAlarmFilter
// 
//	v2.0	|| TC v 3.1.4024.10		|| Transformation to EventLogger TC 3 - in progress
//	v1.2	|| TC v 3.1.4022.25		|| Usuniecie wejscia bEnable
//	v1.1	|| TC v 3.1.4022.25		|| Dodane ACT_EtherCAT_ChangeCounter i Wejscie bEnable
//	v1.0	|| TC v 3.1.4022.20		|| Pierwsza wersja
//==================================================================================================
PROGRAM P_SystemDiag_EventLog
VAR
(*//======================== Checks ===============================
	fbBounds						: FB_AdvancedLogEvent;	// Logowanie wystapienia przekroczenia zakresu indexow
	fbDivDint						: FB_AdvancedLogEvent;	// Logowanie wystapienia proby dzielenia DINT przez 0
	fbDivLInt						: FB_AdvancedLogEvent;	// Logowanie wystapienia proby dzielenia LINT przez 0
	fbDivLReal						: FB_AdvancedLogEvent;	// Logowanie wsytapienia proby dzielenia LREAL przez 0
	fbDivReal						: FB_AdvancedLogEvent;	// Logowanie wystapienia proby dzielenia REAL przez 0
	fbRangeSigned					: FB_AdvancedLogEvent;	// Logowanie wystapienia przekroczenia liczby znakowej
	fbRangeUnsigned					: FB_AdvancedLogEvent;	// Logowanie wystapienia przekroczenia liczby bezznakowej
	
	fbBoundsBlockMessage			: FB_AdvancedLogEvent;	// Logowanie wystapienia przekroczenia zakresu indexow
	fbDivDintBlockMessage			: FB_AdvancedLogEvent;	// Logowanie wystapienia proby dzielenia DINT przez 0
	fbDivLIntBlockMessage			: FB_AdvancedLogEvent;	// Logowanie wystapienia proby dzielenia LINT przez 0
	fbDivLRealBlockMessage			: FB_AdvancedLogEvent;	// Logowanie wsytapienia proby dzielenia LREAL przez 0
	fbDivRealBlockMessage			: FB_AdvancedLogEvent;	// Logowanie wystapienia proby dzielenia REAL przez 0
	fbRangeSignedBlockMessage		: FB_AdvancedLogEvent;	// Logowanie wystapienia przekroczenia liczby znakowej
	fbRangeUnsignedBlockMessage		: FB_AdvancedLogEvent;	// Logowanie wystapienia przekroczenia liczby bezznakowej

//===============================================================
//======================= Persistent ============================
	ftPersistentSave				: F_TRIG;
	fbPersistentEventLoad			: FB_AdvancedLogEvent;
	fbPersistentEventSave			: FB_AdvancedLogEvent;
//===============================================================
//======================== EtherCAT =============================
	bEBusDiagLogPermission			: BOOL	:= TRUE;
	bEBusInitialized				: BOOL;
	iEBusIterator					: INT;
	(*DevDiag SourceID 901*)
	fbEBusDiag						: ARRAY[0..12] OF FB_AdvancedLogEvent;
	fbEtherCATStateChanged			: FB_AdvancedLogEvent;		// ID: 101
	fbEtherCATNotPresent			: FB_AdvancedLogEvent;		// ID: 102
	(*FrmWcState SourceID 902*)
	fbFrmWcDiag						: ARRAY[1..P_EtherCAT_Diag.iNumOfFrames] OF FB_AdvancedLogEvent;
	stFrmDiag						: ARRAY[1..P_EtherCAT_Diag.iNumOfFrames] OF ST_FrmWcDiag;
	fbString						: FB_FormatString;	(*Blok funkcyjny konwertujący FrmWcState na format binarny*)
	tArg							: T_Arg;
	//Filtrowanie zbyt częstego logowania
	fbEBusDiagFilter				: ARRAY[0..12] OF FB_AntiBlinkAlarmFilter;
	fbEBusDiagBlockMessage			: FB_AdvancedLogEvent;
	bFrmDiagLogPermission			: ARRAY[1..P_EtherCAT_Diag.iNumOfFrames] OF BOOL;
	fbFrmDiagFilter					: ARRAY[1..P_EtherCAT_Diag.iNumOfFrames] OF FB_AntiBlinkAlarmFilter;
	fbFrmDiagBlockMessage			: ARRAY[1..P_EtherCAT_Diag.iNumOfFrames] OF FB_AdvancedLogEvent;
//===============================================================
//========================== KBus ===============================
	fbKBusDiag						: ARRAY[0..15] OF FB_AdvancedLogEvent;
	nKbusIterator					: INT;
	bKBusDiagLogPermission			: BOOL := TRUE;
	fbKBusDiagFilter				: ARRAY[0..15] OF FB_AntiBlinkAlarmFilter;
	fbKBusDiagBlockMessage			: FB_AdvancedLogEvent;
//===============================================================
*)
END_VAR

ACT_Checks();
ACT_PersistentLogs();
ACT_EtherCAT_Diag();
ACT_EtherCAT_ChangeCounter();
// ACT_KBus(); 
//===============================================================
//==================== In preparation ===========================
//======================== TaskInfo =============================
//===============================================================

ACTION ACT_Checks:
(*fbBounds(
	bSetEvent		:= P_Checks.bCheckBounds,
	eEventClass 	:= TCEVENTCLASS_ALARM,
	bQuit			:= FALSE, 
	udiSourceID		:= 905, 
	udiEventID		:= 1);

fbDivDint(
	bSetEvent		:= P_Checks.bCheckDivDint,
	eEventClass 	:= TCEVENTCLASS_ALARM,
	bQuit			:= FALSE, 
	udiSourceID		:= 905, 
	udiEventID		:= 2);
	
fbDivLInt(
	bSetEvent		:= P_Checks.bCheckDivLInt,
	eEventClass 	:= TCEVENTCLASS_ALARM,
	bQuit			:= FALSE, 
	udiSourceID		:= 905, 
	udiEventID		:= 3);
	
fbDivLReal(
	bSetEvent		:= P_Checks.bCheckDivLReal,
	eEventClass 	:= TCEVENTCLASS_ALARM,
	bQuit			:= FALSE, 
	udiSourceID		:= 905, 
	udiEventID		:= 4);
	
fbDivReal(
	bSetEvent		:= P_Checks.bCheckDivReal,
	eEventClass 	:= TCEVENTCLASS_ALARM,
	bQuit			:= FALSE, 
	udiSourceID		:= 905, 
	udiEventID		:= 5);
	
fbRangeSigned(
	bSetEvent		:= P_Checks.bCheckRangeSigned,
	eEventClass 	:= TCEVENTCLASS_ALARM,
	bQuit			:= FALSE, 
	udiSourceID		:= 905, 
	udiEventID		:= 6);
	
fbRangeUnsigned(
	bSetEvent		:= P_Checks.bCheckRangeUnsigned,
	eEventClass 	:= TCEVENTCLASS_ALARM,
	bQuit			:= FALSE, 
	udiSourceID		:= 905, 
	udiEventID		:= 7);
	*)
END_ACTION

ACTION ACT_EtherCAT_ChangeCounter:
(*fbEtherCATStateChanged(	bSetEvent		:= P_EtherCAT_ChangeCounter.bAbnormalStateChangeCounterChanged, 
						bQuit			:= FALSE, 
						udiSourceID		:= 901, 
						udiEventID		:= 101, 
						sFormat			:= '%d', 
						eEventClass		:= TCEVENTCLASS_ALARM, 
						pDataAddress	:= ADR(P_EtherCAT_ChangeCounter.wAbnormalStateChangeCounterPosition), 
						udiDataLenght	:= SIZEOF(P_EtherCAT_ChangeCounter.wAbnormalStateChangeCounterPosition));

fbEtherCATNotPresent(	bSetEvent		:= P_EtherCAT_ChangeCounter.bPresentStateChangeCounterChanged, 
						bQuit			:= FALSE, 
						udiSourceID		:= 901, 
						udiEventID		:= 102, 
						sFormat			:= '%d', 
						eEventClass		:= TCEVENTCLASS_ALARM, 
						pDataAddress	:= ADR(P_EtherCAT_ChangeCounter.wPresentStateChangeCounterPosition), 
						udiDataLenght	:= SIZEOF(P_EtherCAT_ChangeCounter.wPresentStateChangeCounterPosition));
*)
END_ACTION

ACTION ACT_EtherCAT_Diag:
(*// Wstępne zezwolenie na logowanie alarmów
IF NOT bEBusInitialized THEN
	FOR iEBusIterator := 1 TO P_EtherCAT_Diag.iNumOfFrames DO
		bFrmDiagLogPermission[iEBusIterator]	:= TRUE;
	END_FOR
	bEBusInitialized					:= TRUE;
END_IF

// DevState
FOR iEBusIterator := 0 TO 12 DO
	fbEBusDiag[iEBusIterator](
						bSetEvent		:= GETBIT32(P_EtherCAT_Diag.uiDevState,INT_TO_SINT(iEBusIterator)) AND bEBusDiagLogPermission,
						eEventClass 	:= TCEVENTCLASS_ALARM,
						bQuit			:= FALSE,
						udiSourceID		:= 901,
						udiEventID		:= INT_TO_UDINT(iEBusIterator + 1));
END_FOR

// FrmWcState
FOR iEBusIterator := 1 TO P_EtherCAT_Diag.iNumOfFrames DO
	stFrmDiag[iEBusIterator].iNum		:= iEBusIterator;
	IF P_EtherCAT_Diag.uiFrmWcState[iEBusIterator] <> 0 THEN
		tArg.cbLen						:= SIZEOF(P_EtherCAT_Diag.uiFrmWcState[iEBusIterator]);
		tArg.eType						:= ARGTYPE_UINT;
		tArg.pData						:= ADR(P_EtherCAT_Diag.uiFrmWcState[iEBusIterator]);
		fbString(sFormat := '%b', arg1 := tArg);
		stFrmDiag[iEBusIterator].sBin 	:= fbString.sOut;
	END_IF
	fbFrmWcDiag[iEBusIterator](
						bSetEvent		:= NOT(P_EtherCAT_Diag.uiFrmWcState[iEBusIterator] = 0) AND bFrmDiagLogPermission[iEBusIterator],
						eEventClass 	:= TCEVENTCLASS_ALARM,
						bQuit			:= FALSE, 
						udiSourceID		:= 902,
						udiEventID		:= INT_TO_UDINT(iEBusIterator),
						sFormat			:= '%d%s',
						pDataAddress	:= ADR(stFrmDiag[iEBusIterator]),
						udiDataLenght	:= SIZEOF(stFrmDiag[iEBusIterator]) );
END_FOR
*)
END_ACTION

ACTION ACT_KBus:
(*// Send errors to event logger
FOR nKbusIterator := 0 TO 15 DO
	fbKBusDiag[nKbusIterator](
		bSetEvent					:= GETBIT32(P_KBus.uiKbusState,INT_TO_SINT(nKbusIterator)) AND bKBusDiagLogPermission,	// maskowanie bitów
		eEventClass 				:= TCEVENTCLASS_ALARM,
		bQuit						:= FALSE,
		udiSourceID					:= 904,
		udiEventID					:= INT_TO_UDINT(nKbusIterator),
		sFormat						:= '');
	// Filter
	fbKBusDiagFilter[nKbusIterator](bEvent := GETBIT32(P_KBus.uiKbusState,INT_TO_SINT(nKbusIterator)),
		tTime						:= T#1S,
		uiLimit						:= 2,
		bPermission					:= bKBusDiagLogPermission);
END_FOR

fbKBusDiagBlockMessage(
	bSetEvent						:= NOT bKBusDiagLogPermission,
	eEventClass 					:= TCEVENTCLASS_MESSAGE,
	bQuit							:= FALSE , 
	udiSourceID						:= 904, 
	udiEventID						:= 100);
	*)
END_ACTION

ACTION ACT_PersistentLogs:
(*IF _TaskInfo[1].FirstCycle THEN
	fbPersistentEventLoad.bSetEvent 			:= TRUE;
	IF _AppInfo.BootDataLoaded AND _AppInfo.OldBootData = FALSE THEN 	// wczytano poprawnie zmienne nieulotne
		fbPersistentEventLoad.udiEventID		:= 1;
		fbPersistentEventLoad.eEventClass		:= TCEVENTCLASS_MESSAGE;
	ELSIF _AppInfo.BootDataLoaded AND _AppInfo.OldBootData THEN 		// wczytano zmienne z kopii
		fbPersistentEventLoad.udiEventID		:= 2;
		fbPersistentEventLoad.eEventClass		:= TCEVENTCLASS_WARNING;
	ELSE //blad wczytania zmiennych
		fbPersistentEventLoad.udiEventID		:= 3;
		fbPersistentEventLoad.eEventClass		:= TCEVENTCLASS_ALARM;
	END_IF
ELSE
	//gdy nie wczytało zmiennych nieulotnych to wyswietlaj ostrzezenie w eventach aktywnych
	IF NOT (_AppInfo.BootDataLoaded = FALSE AND _AppInfo.OldBootData = FALSE) THEN
		fbPersistentEventLoad.bSetEvent			:= FALSE;
	END_IF
END_IF

fbPersistentEventLoad(udiSourceID := 900);

ftPersistentSave (CLK := P_Persistent.fbWritePersistentData.BUSY);
IF ftPersistentSave.Q THEN
	fbPersistentEventSave.bSetEvent 			:= TRUE;
	IF P_Persistent.fbWritePersistentData.ERR THEN
		fbPersistentEventSave.sFormat 			:= '%d';
		fbPersistentEventSave.udiEventID		:= 11;
		fbPersistentEventSave.eEventClass		:= TCEVENTCLASS_ALARM;
		fbPersistentEventSave.pDataAddress		:= ADR(P_Persistent.fbWritePersistentData.ERRID);
		fbPersistentEventSave.udiDataLenght		:= SIZEOF(P_Persistent.fbWritePersistentData.ERRID);
	ELSE
		fbPersistentEventSave.sFormat			:= '';
		fbPersistentEventSave.udiEventID		:= 10;
		fbPersistentEventSave.eEventClass		:= TCEVENTCLASS_MESSAGE;
	END_IF
ELSE
	fbPersistentEventSave.bSetEvent				:= FALSE;
END_IF

fbPersistentEventSave(udiSourceID:= 900);
*)
END_ACTION

END_PROGRAM

// ---- POUs/POUsDiagnostics/FB/FB_AntiBlinkAlarmFilter.TcPOU
//==================================================================================================
//							Beckhoff Automation Poland
//								FB_AntiBlinkAlarmFilter
//									20.12.2016
//				Blok służący do wyłączania logowania zdarzeń które pojawiają się zbyt często
// 	v1.0 || TC v 3.1.4020.28 || - pierwsza wersja
//==================================================================================================
FUNCTION_BLOCK FB_AntiBlinkAlarmFilter
VAR_INPUT
	bEvent			: BOOL;		// Status zdarzenia
	tTime			: TIME;		// Zadane okno czasowe
	uiLimit			: UINT;		// Maksymalna liczba zdarzeń jaka może się pojawić w oknie czasowym
END_VAR
VAR_IN_OUT
	bPermission		: BOOL;		// Flaga zezwolenia na logowanie zdarzeń
END_VAR
VAR
	tStartTime		: TIME;		// Zmienna przechowująca czas rozpoczęcia zliczania
	uiActCount		: UINT;		// Aktualna wartość licznika
	rtEdge			: R_TRIG;	// Zbocze narastające
END_VAR

rtEdge(CLK:=bEvent);
IF rtEdge.Q THEN							// Blok podejmuje akcję w przypadku wystapienia zdarzenia
	IF uiActCount = 0 THEN	
		tStartTime		:= TIME();			// W przypadku gdy licznik wynosi zero, zapisywany jest czas rozpoczęcia zliczania
	END_IF
	uiActCount			:= uiActCount + 1;	// Inkrementacja licznika liczby zdarzeń
	IF uiActcount >= uiLimit THEN			// W przypadku gdy liczba zdarzeń osiągnie zadany limit, sprawdzany jest czas w jakim one wystapiły. Jeśli czas jest większy niż dopuszczalny, resetowana jest flaga zezwolenia
		IF TIME() - tStartTime < tTime THEN
			bPermission	:= FALSE;		
		END_IF
		uiActCount 		:= 0;
	END_IF
	IF NOT bPermission THEN
		uiActCount		:= 0;
	END_IF
END_IF;

END_FUNCTION_BLOCK

// ---- POUs/P_EventLogger_Simple.TcPOU
PROGRAM P_EventLogger_Simple
VAR
	rtMessage 			: ARRAY [1..GVL_EventLogger_Simple.nMaxNumMessages] OF R_TRIG;
	rtWarning 			: ARRAY [1..GVL_EventLogger_Simple.nMaxNumWarnings] OF R_TRIG;
	rtError 			: ARRAY [1..GVL_EventLogger_Simple.nMaxNumErrors] OF R_TRIG;
	ftError 			: ARRAY [1..GVL_EventLogger_Simple.nMaxNumErrors] OF F_TRIG;
	rtErrorConfirm		: ARRAY [1..GVL_EventLogger_Simple.nMaxNumErrors] OF R_TRIG;
	
	fbTcMessage 		: FB_TcMessage;
	fbTcWarning 		: FB_TcMessage;
	fbTcError 			: ARRAY [1..GVL_EventLogger_Simple.nMaxNumErrors] OF FB_TcAlarm;
	
	idx					: UDINT;
	bAlarmsInitialized	: BOOL;
END_VAR

// Messages
FOR idx := 1 TO GVL_EventLogger_Simple.nMaxNumMessages DO	
	rtMessage[idx](CLK := GVL_EventLogger_Simple.arrMessageTriggers[idx]);
	IF rtMessage[idx].Q THEN
		GVL_EventLogger_Simple.arrMessageTriggers[idx] := FALSE; // auto clear
		fbTcMessage.Create(TC_EVENT_CLASSES.MyMessages, idx, TcEventSeverity.Verbose, 0);
		fbTcMessage.Send(0);
	END_IF
END_FOR

// Warnings
FOR idx := 1 TO GVL_EventLogger_Simple.nMaxNumWarnings DO	
	rtWarning[idx](CLK := GVL_EventLogger_Simple.arrWarningTriggers[idx]);
	IF rtWarning[idx].Q THEN
		GVL_EventLogger_Simple.arrWarningTriggers[idx] := FALSE; // auto clear
		fbTcWarning.Create(TC_EVENT_CLASSES.MyWarnings, idx, TcEventSeverity.Warning, 0);
		fbTcWarning.Send(0);
	END_IF
END_FOR

// Alarms
IF NOT bAlarmsInitialized THEN
	bAlarmsInitialized := TRUE;
	FOR idx := 1 TO GVL_EventLogger_Simple.nMaxNumErrors DO	
		fbTcError[idx].Create(TC_EVENT_CLASSES.MyErrors, idx, TcEventSeverity.Error, TRUE, 0);
	END_FOR	
END_IF

FOR idx := 1 TO GVL_EventLogger_Simple.nMaxNumErrors DO	
	rtError[idx](CLK := GVL_EventLogger_Simple.arrErrorTriggers[idx]);
	ftError[idx](CLK := GVL_EventLogger_Simple.arrErrorTriggers[idx]);
	rtErrorConfirm[idx](CLK := GVL_EventLogger_Simple.arrErrorConfirmations[idx]);
	IF rtError[idx].Q THEN
		fbTcError[idx].Raise(0);
	END_IF
	IF ftError[idx].Q THEN
		fbTcError[idx].Clear(0, FALSE);
	END_IF
	IF rtErrorConfirm[idx].Q THEN
		GVL_EventLogger_Simple.arrErrorConfirmations[idx] := FALSE; // auto clear
		fbTcError[idx].Confirm(0);
	END_IF	
END_FOR

END_PROGRAM

// ---- POUs/P_ErrorCollection.TcPOU
//==================================================================================================
//							Beckhoff Automation Poland
//									2.11.2018
//	Place to collect all module error, warning, ready etc flags. Here You can mute errors also.
// 
//	v1.0 	|| TC v 3.1.4022.25 		|| Pierwsza wersja
//==================================================================================================
PROGRAM P_ErrorCollection
VAR
	bOK										: BOOL;
	bWarning								: BOOL;
	bError									: BOOL;
	bFatalError								: BOOL;
END_VAR

bError := P_SystemDiagnostics.bError OR P_Template_SAFETY.bError; // And more....
// Collect flags - real
bWarning  								:= bWarning; 										// Collection
bError  								:= bError; 											// Collection
bFatalError  							:= bFatalError; 									// Collection
bOk										:= NOT (bWarning OR bError OR bFatalError);
// Pass to global, add mute if neccesary
GVL.bGeneralWarning  					:= bWarning;										// Pass
GVL.bGeneralError  						:= bError AND NOT GVL.bMuteGeneralError;			// Pass and mute
GVL.bGeneralFatalError  				:= bFatalError AND NOT GVL.bMuteGeneralFatalError;	// Pass and mute
GVL.bGeneralOK 							:= NOT GVL.bGeneralWarning OR GVL.bGeneralError OR GVL.bGeneralFatalError;
// Machine units ready flag
GVL.bAllUnitsReady 						:= NOT (P_Template.bError (*OR P_Template_CAM.bError*));	// All units
// After fatal error and auto mode machine reset is required
GVL.bRestartRequired					R= NOT GVL.bGeneralFatalError;
GVL.bRestartRequired					S= GVL.bGeneralFatalError AND (GVL_Machine.eMode = E_MachineMode.eAutomatic);

END_PROGRAM

// ---- POUs/P_Template_SAFETY.TcPOU
PROGRAM P_Template_SAFETY
VAR_INPUT
	eMachineMode							: E_MachineMode; 		// Machine mode
	eMachineCommand							: E_MachineCommand; 	// Command from top level state program
END_VAR
VAR_OUTPUT
	eMachineState							: E_MachineState;
  	bError									: BOOL;
END_VAR
VAR
	// INPUTS
	bResetBusy								: BOOL;
	// OUTPUTS
	bResetCMD								: BOOL;
	// FBs
	rtRestart								: R_TRIG;
	rtReset									: R_TRIG;
	ftFinish								: F_TRIG;
	bSTOStatus								: BOOL;
	bSOSStatus								: BOOL;
	bAllAxisInSafeState						: BOOL;
	bAllAxisReady							: BOOL;
END_VAR

// =================== Inputs ===================
// Read input signals
Act_InUpdate();

// Error collection
Act_Error();
// ==============================================
rtReset(CLK:= eMachineCommand = E_MachineCommand.eReset, Q=> );
rtRestart(CLK:= eMachineCommand = E_MachineCommand.eRestart, Q=> );
ftFinish(CLK:= bResetBusy, Q=> );

IF bError THEN
	eMachineState								:= E_MachineState.eError;
END_IF

IF rtRestart.Q THEN
	eMachineState								:= E_MachineState.eRestarting;
	bResetCMD									:= TRUE;
END_IF

IF rtReset.Q THEN
	eMachineState								:= E_MachineState.eReseting;
	bResetCMD									:= TRUE;
END_IF

IF ftFinish.Q THEN
	eMachineState								:= E_MachineState.eRunning;
	bResetCMD									:= FALSE;
END_IF

// =================== Outputs ==================
Act_OutUpdate();
// ==============================================

ACTION Act_Error:
// Program summary error
bError 							:= 	(GVL_IO.dwAXErrors OR GVL_IO.dwGroupErrors) <> 0;
// OR bError 							:= GVL_IO.bSAFETY_Error;
END_ACTION

ACTION Act_InUpdate:
bResetBusy 						:= GVL_IO.bSAFETY_ResetBusy;
bSTOStatus  					:= GVL_IO.dwAXStatesSTO = 2#11_1111;
bSOSStatus  					:= GVL_IO.dwAXStatesSOS = 2#1111;
bAllAxisInSafeState  			:= (GVL_IO.dwAXStatesSTO OR GVL_IO.dwAXStatesSOS) = 2#11_1111;
bAllAxisReady 					:= (GVL_IO.dwAXStatesSTO OR GVL_IO.dwAXStatesSOS) = 0;
END_ACTION

ACTION Act_OutUpdate:
GVL_IO.bSAFETY_ResetCMD 		:= bResetCMD;
END_ACTION

END_PROGRAM

// ---- POUs/P_Template.TcPOU
PROGRAM P_Template
VAR_INPUT
	eMachineMode							: E_MachineMode; 		// Machine mode
	eMachineCommand							: E_MachineCommand; 	// Command from top level state program
END_VAR
VAR_OUTPUT
	eMachineState							: E_MachineState;
  	bError									: BOOL;
END_VAR
VAR_IN_OUT
	Axis1									: AXIS_REF;
END_VAR
VAR
	// INPUTS
	bIn1									: BOOL;
	// OUTPUTS
	bOut1									: BOOL;	
	// Local
	iStepInit								: INT; 					// CASE inicjalizacji
	iStepAuto					 			: INT;
	// HMI Maintenance 
	
	// FBs Axis Online
	fbAxis1									: FB_McAxisOnlineAX5000;
	stAxis1									: ST_McAxisOnline;
END_VAR

// Always clear command in active step

// Read input signals
Act_InUpdate();

// ====================================================
// FBs CALL

// Monitoring
Act_Monitoring();
	
// Error collection
Act_Error();

// SAFETY CALL 
// Abort CMD is avaliable in each mode in each state except Aborted - because in it is already safe, we don't want to repat CMD in loop
IF eMachineCommand = E_MachineCommand.eAbort AND eMachineState <> E_MachineState.eAborted THEN
	eMachineState								:= E_MachineState.eAborting;
END_IF

// Machine mode change over
CASE eMachineMode OF
	
	E_MachineMode.eInitialization:
		; // Do nothing
	
	E_MachineMode.eAutomatic:
		Act_ModeAutomatic();
		
	E_MachineMode.eManual:
		Act_ModeManual();	
		
	E_MachineMode.eMaintenance:
		Act_ModeMaintenance();	
		
END_CASE

// Call Axis online FBs
fbAxis1(stMcAxisOnline:= stAxis1, Axis:= Axis1);

// Write outputs
Act_OutUpdate();

ACTION Act_Error:
// Program summary error
bError := 	bError; // ie. Init Error
			// OR axis error
			// OR item error
END_ACTION

ACTION Act_InUpdate:
bIn1 := TRUE; // Assign, filters, conditions, scaling etc
END_ACTION

ACTION Act_ModeAutomatic:
// State Machine
CASE eMachineState OF

	E_MachineState.eIdle:
	
		// Idle - there should be done background initialization. We do it just once.
		// ====================================================
		// There should be main code
		// i.e. CASE iStepInit OF	
		// ====================================================
		// Allow for stop only if conditions are true - in this step we can wait without an error	
		IF TRUE (* condition *) AND eMachineCommand = E_MachineCommand.eStop THEN
			eMachineState 						:= E_MachineState.eStopped;
		END_IF
		
		IF bError THEN
			eMachineState 						:= E_MachineState.eError;
		END_IF
		
	E_MachineState.eStopping:

		// Stopping action in our sample - empty instruction and go to Stopped
		// In real app we should execute CMD and wait for finish (all items) - done, abort or error
		// In this phase we don't look into error
		IF TRUE (* condition *) THEN
			eMachineState 						:= E_MachineState.eStopped;
		END_IF
		
		// Alternative - in some apps it's neccasary to go into an error as soon as first error occured - You have to decide
		
	E_MachineState.eStopped:

		// In this step we just wait for CMD or for Error
		IF eMachineCommand = E_MachineCommand.eRun THEN
			eMachineState 						:= E_MachineState.eStarting;
		END_IF

		IF bError THEN
			eMachineState 						:= E_MachineState.eError;
		END_IF

	E_MachineState.eStarting:

		// Starting action in our sample - empty instruction and go to Running
		// It can be init, monitoring etc, in some apps enable drives cmd is here
		IF TRUE (* condition *) THEN
			eMachineState 						:= E_MachineState.eRunning;
		END_IF
		
	E_MachineState.eRunning:

		// ====================================================
		// There should be main code
		// i.e. CASE iStepAuto OF
		// ====================================================
		IF eMachineCommand = E_MachineCommand.eStop OR bError THEN
			eMachineState 						:= E_MachineState.eStopping;
		END_IF

	E_MachineState.eAborting:

		// Stop and reset everything - usually SAFETY function
		IF TRUE (* condition *) THEN
			eMachineState 						:= E_MachineState.eAborted;
		END_IF
		
	E_MachineState.eAborted:
	
		IF eMachineCommand = E_MachineCommand.eReset THEN
			eMachineState 						:= E_MachineState.eReseting;
		END_IF
		
		IF bError THEN
			eMachineState 						:= E_MachineState.eError;
		END_IF

	E_MachineState.eError:

		// ====================================================
		// Two types of error:
		// 1. 'Small/soft' Error - fix a problem and go to stop
		// 2. 'Serious/hard' Error - there is a need of restart everything, if there is a sequence - reset it too - fix a problem and go to init
		// ====================================================
		IF eMachineCommand = E_MachineCommand.eReset THEN
			eMachineState 						:= E_MachineState.eReseting;
		END_IF
		
		IF eMachineCommand = E_MachineCommand.eRestart THEN
			eMachineState 						:= E_MachineState.eRestarting;
		END_IF

	E_MachineState.eReseting:

		// ====================================================
		//'Small/soft' Error - fix a problem and go to stop
		// Reset drives only when it is necessary
		// ====================================================
		// Check if axis errors cleared
		IF TRUE (*NOT bAxisError AND NOT other errors *) THEN
			eMachineState  						:= E_MachineState.eStopping;
		END_IF
		
		// In this state we don't monitor general Error, just reset procedure error		
		IF FALSE (* bResetError *) THEN
			eMachineState  						:= E_MachineState.eError;
		END_IF
		
	E_MachineState.eRestarting:

		// ====================================================
		// 'Serious/hard' Error - there is a need of restart everything, if there is a sequence - reset it too - fix a problem and go to init
		// Reset drives only when it is necessary
		// ====================================================
		// Check if axis errors cleared
		IF TRUE (*NOT bAxisError AND NOT other errors *) THEN
			eMachineState  						:= E_MachineState.eIdle;
		END_IF
				
		// In this state we don't monitor general Error, just reset procedure error		
		IF FALSE (* bResetError *) THEN
			eMachineState  						:= E_MachineState.eError;
		END_IF
		
END_CASE
END_ACTION

ACTION Act_ModeMaintenance:
// State Machine
CASE eMachineState OF

	E_MachineState.eIdle, E_MachineState.eStopping, E_MachineState.eStopped, E_MachineState.eStarting:
	
		// ====================================================
		// There should be main code
		// i.e. CASE iStepInit OF	
		// ====================================================
		// Allow for stop only if conditions are true - in this step we can wait without an error	
		IF TRUE (* condition *) AND eMachineCommand = E_MachineCommand.eRun THEN
			eMachineState 						:= E_MachineState.eRunning;
		END_IF

	E_MachineState.eRunning:

		// ====================================================
		// HMI control
		// There should be main code,
		// i.e. CASE iStepAuto OF
		// ====================================================
		IF eMachineCommand = E_MachineCommand.eStop THEN
			eMachineState 						:= E_MachineState.eStopping;
		END_IF

	E_MachineState.eAborting:

		// Stop and reset everything - usually SAFETY function
		IF TRUE (* condition *) THEN
			eMachineState 						:= E_MachineState.eAborted;
		END_IF
		
	E_MachineState.eAborted:

		IF eMachineCommand = E_MachineCommand.eReset THEN
			eMachineState 						:= E_MachineState.eReseting;
		END_IF

	E_MachineState.eRestarting, E_MachineState.eReseting, E_MachineState.eError:

			;// Unused

END_CASE
END_ACTION

ACTION Act_ModeManual:

END_ACTION

ACTION Act_Monitoring:
// Ustawianie flag, monitoring kolizjii, watchdogi, jazdy po krzywce itp
;
END_ACTION

ACTION Act_OutUpdate:
;
END_ACTION

END_PROGRAM

// ---- POUs/POUsAxisOnline/AX5000/FB_McAxisOnlineAX5000.TcPOU
//==================================================================================================
//							Beckhoff Automation Poland
//									7.12.2018
//	Wszystkomajacy blok funkcyjny do sterowania osia, 
//	wymagane biblioteki: Tc2_EtherCAT, Tc2_Drive, Tc2_MC2_Drive, Tc2_MC2, Tc2_Utilities
//  v1.2	|| TC v 3.1.4022.27		|| - dodane opisy bledow w formie zmiennych typu string
// 	v1.1 	|| TC v 3.1.4022.20	 	|| - ACT_MotorMonitoring - only for real axis
// 	v1.0 	|| TC v 3.1.4022.16	 	|| - first edition
//==================================================================================================
{attribute 'reflection'}
FUNCTION_BLOCK FB_McAxisOnlineAX5000
VAR_IN_OUT
	stMcAxisOnline						: ST_McAxisOnline;
	Axis								: AXIS_REF;
END_VAR
VAR
	mcPower								: MC_Power;
	mcStop								: MC_Stop;
	mcHalt								: MC_Halt;
	mcStopSS1							: MC_Stop;
	mcStopSS2							: MC_Stop;
	mcReset								: MC_Reset;
	mcHome								: MC_Home;
	mcSetPosition						: MC_SetPosition;
	fbSetPositionOffset					: FB_SetPositionOffset;
	mcJog								: MC_Jog;

	mcMoveAbsolute						: MC_MoveAbsolute;
	mcMoveRelative						: MC_MoveRelative;
	mcMoveVelocity						: MC_MoveVelocity;
	mcMoveModulo						: MC_MoveModulo;
	mcMoveAbsolute2						: MC_MoveAbsolute;
	mcMoveRelative2						: MC_MoveRelative;
	mcMoveVelocity2						: MC_MoveVelocity;
	mcMoveModulo2						: MC_MoveModulo;

	fbMotorMonitoring					: FB_MotorMonitoringAX5000;
	fbHoldingBrakeCtrl					: FB_HoldingBrakeCtrlAX5000;
	fbNcLimitSwitch						: FB_NcSWLimitSwitchCtrl;
	tonGetDriveDiag						: TON;
	fbReadChannelErrorCode				: FB_AxisDiag;
	
	mcReadDriveAddress					: MC_ReadDriveAddress;
	mcReadParameterSet					: MC_ReadParameterSet;
	fbGetDriveRef						: FB_GetDriveRef;

	// Internal
	bInitialized						: BOOL;
			
	// Initialization
	iInitStep							: INT;
	bInitializationError				: BOOL;
	wInitializationErrorCounter			: WORD;
	bDriveAddressReady					: BOOL;
	bDriveRefReady						: BOOL;
	bReadParameterSetReady				: BOOL;
	tonDelay							: TON;
	// Re init
	udiOnlineChangeCntOld				: UDINT;
	bOnlineChangeDetected				: BOOL;
	bReInit								: BOOL;
	bReInitialized						: BOOL;
	bReInitializationError				: BOOL;
	// Axis diag struct
	stAX5000Diag						: ST_AX5000Diag;
	{attribute 'instance-path'}
	{attribute 'noinit'}
	sInstancePath						: STRING;
END_VAR

// Device dependent initialization 
ACT_Initialization();
// Device independent commands, mostly NC 
ACT_States();
ACT_SWLimitSwitch();
ACT_Stop();
ACT_Power();
ACT_Homing();
ACT_Jog();
ACT_Move();
ACT_ResetAndDiag();
ACT_SetPosition();
// Device dependent commands
// Motor monitoring possible only with real axis
IF NOT Axis.Status.OpMode.SimulationAxis THEN
	ACT_MotorMonitoring();
END_IF
// Device dependent commands, possible only on real axis after complete initialization
IF bInitialized AND NOT Axis.Status.OpMode.SimulationAxis THEN
	ACT_SetPositionIO();
	ACT_HoldingBrakeCtrl();
END_IF

// Device independent error collection
ACT_ErrorCollection();

ACTION ACT_ErrorCollection:
// Error flags
stMcAxisOnline.stError.bDriveError					:= Axis.Status.DriveDeviceError;

stMcAxisOnline.stError.bNcError						:= Axis.Status.Error;

stMcAxisOnline.stError.bFBError						:= stMcAxisOnline.mcPower.bError OR stMcAxisOnline.mcReset.bError OR stMcAxisOnline.mcHome.bError OR stMcAxisOnline.mcJog.bError
													OR stMcAxisOnline.mcHalt.bError OR stMcAxisOnline.mcStop.bError OR stMcAxisOnline.mcSS1.bError OR stMcAxisOnline.mcSS2.bError
													OR stMcAxisOnline.mcMoveAbsolute.bError OR stMcAxisOnline.mcMoveRelative.bError OR stMcAxisOnline.mcMoveVelocity.bError OR stMcAxisOnline.mcMoveModulo.bError
													OR stMcAxisOnline.mcMoveAbsolute2.bError OR stMcAxisOnline.mcMoveRelative2.bError OR stMcAxisOnline.mcMoveVelocity2.bError OR stMcAxisOnline.mcMoveModulo2.bError
													OR stMcAxisOnline.stNcLimitSwitch.bError OR stMcAxisOnline.mcSetPosition.bError;
									
stMcAxisOnline.stError.bCommunicationError			:= stMcAxisOnline.stChannelErrorCode.bError OR stMcAxisOnline.stSetPositionOffset.bError OR stMcAxisOnline.stMotorMonitoring.bError OR stMcAxisOnline.stHoldingBrake.bError;

stMcAxisOnline.stError.bError						:= stMcAxisOnline.stError.bDriveError OR stMcAxisOnline.stError.bNcError OR stMcAxisOnline.stError.bFBError OR stMcAxisOnline.stError.bCommunicationError;
stMcAxisOnline.bError								:= stMcAxisOnline.stError.bError; // Forward one stage up

// Error codes
stMcAxisOnline.stError.uiDriveErrorID 				:= stMcAxisOnline.stChannelErrorCode.uiChannelErrorCode;
stMcAxisOnline.stError.uiDriveErrorIDHex 			:= stMcAxisOnline.stChannelErrorCode.uiChannelErrorCodeHex;

stMcAxisOnline.stError.udiNcErrorID 				:= Axis.Status.ErrorID;
stMcAxisOnline.stError.udiNcErrorIDHex 				:= Axis.Status.ErrorID;
	

stMcAxisOnline.stError.udiFBErrorID 				:= 	stMcAxisOnline.mcPower.udiErrorID + 
														stMcAxisOnline.mcReset.udiErrorID + 
														stMcAxisOnline.mcHome.udiErrorID + 
														stMcAxisOnline.mcJog.udiErrorID +
														stMcAxisOnline.mcHalt.udiErrorID + 
														stMcAxisOnline.mcStop.udiErrorID + 
														stMcAxisOnline.mcSS1.udiErrorID + 
														stMcAxisOnline.mcSS2.udiErrorID +
														stMcAxisOnline.mcMoveAbsolute.udiErrorID + 
														stMcAxisOnline.mcMoveRelative.udiErrorID + 
														stMcAxisOnline.mcMoveVelocity.udiErrorID + 
														stMcAxisOnline.mcMoveModulo.udiErrorID +
														stMcAxisOnline.mcMoveAbsolute2.udiErrorID + 
														stMcAxisOnline.mcMoveRelative2.udiErrorID + 
														stMcAxisOnline.mcMoveVelocity2.udiErrorID + 
														stMcAxisOnline.mcMoveModulo2.udiErrorID +
														stMcAxisOnline.stNcLimitSwitch.udiErrorID + 
														stMcAxisOnline.mcSetPosition.udiErrorID;

stMcAxisOnline.stError.udiFBErrorIDHex 				:= stMcAxisOnline.stError.udiFBErrorID;

stMcAxisOnline.stError.udiErrorID					:= stMcAxisOnline.stSetPositionOffset.udiErrorID;
stMcAxisOnline.stError.uiAdsErrorID					:= stMcAxisOnline.stChannelErrorCode.uiAdsErrId + stMcAxisOnline.stMotorMonitoring.uiAdsErrId + stMcAxisOnline.stHoldingBrake.uiAdsErrId;
stMcAxisOnline.stError.uiSecErrorID					:= stMcAxisOnline.stChannelErrorCode.uiSecErrId + stMcAxisOnline.stMotorMonitoring.uiSecErrId + stMcAxisOnline.stHoldingBrake.uiSecErrId;

stMcAxisOnline.stError.sNcError						:= F_AxErrMsg(stMcAxisOnline.stError.udiNcErrorID);
stMcAxisOnline.stError.sDriveError					:= F_AX5xErrMsg(stMcAxisOnline.stError.uiDriveErrorID);
END_ACTION

ACTION ACT_HoldingBrakeCtrl:
fbHoldingBrakeCtrl(
					bForceLock			:= stMcAxisOnline.stHoldingBrake.bForceLock,
					bForceUnlock		:= stMcAxisOnline.stHoldingBrake.bForceUnlock,
					bBusy				=> stMcAxisOnline.stHoldingBrake.bBusy,
					bError				=> stMcAxisOnline.stHoldingBrake.bError,
					iAdsErrId			=> stMcAxisOnline.stHoldingBrake.uiAdsErrId,
					iSecErrId			=>stMcAxisOnline.stHoldingBrake.uiSecErrId , 
					Axis				:= Axis );
END_ACTION

ACTION ACT_Homing:
mcHome(		Axis						:= Axis,
			Execute						:= stMcAxisOnline.mcHome.bExecute,
			Position					:= stMcAxisOnline.mcHome.lrPosition,
			HomingMode					:= stMcAxisOnline.mcHome.eHomingMode,
			BufferMode					:= stMcAxisOnline.mcHome.eBufferMode,
			Options						:= stMcAxisOnline.mcHome.stOptions,
			bCalibrationCam				:= stMcAxisOnline.mcHome.bCalibrationCam,
			Done						=> stMcAxisOnline.mcHome.bDone,
			Busy						=> stMcAxisOnline.mcHome.bBusy,
			Active						=> stMcAxisOnline.mcHome.bActive,
			CommandAborted				=> stMcAxisOnline.mcHome.bCommandAborted,
			Error						=> stMcAxisOnline.mcHome.bError,
			ErrorID						=> stMcAxisOnline.mcHome.udiErrorID);
END_ACTION

ACTION ACT_Initialization:
// bInitialized flag is set just once. 
// bReInitialized ise set each time we do online change or request reinit operation
// bDriveAddressReady, bReadParameterSetReady, bDriveRefReady - set just once after successed read

// Online change detection
bOnlineChangeDetected					:= udiOnlineChangeCntOld <> _AppInfo.OnlineChangeCnt;
udiOnlineChangeCntOld 					:= _AppInfo.OnlineChangeCnt;
// Reset init
IF bReInit OR bOnlineChangeDetected THEN
	iInitStep							:= 0;
END_IF

//Initialization process
CASE iInitStep OF
	0:	// Read Drive Address
		
		stMcAxisOnline.mcReadDriveAddress.bExecute	:=	 TRUE;
		iInitStep						:= iInitStep + 10;
		
	10: // Wait for data
	
		IF NOT stMcAxisOnline.mcReadDriveAddress.bBusy THEN
			stMcAxisOnline.mcReadDriveAddress.bExecute	:=	 FALSE;
			IF stMcAxisOnline.mcReadDriveAddress.bDone THEN
				iInitStep 				:= iInitStep + 10;
				bDriveAddressReady 		:= TRUE;
			ELSE
				iInitStep 				:= 1000;		// Error step
			END_IF
		END_IF
		
	20:	// Read Parameter Set
		
		stMcAxisOnline.mcReadParameterSet.bExecute		:=	 TRUE;
		iInitStep						:= iInitStep + 10;
		
	30: // Wait for data
	
		IF NOT stMcAxisOnline.mcReadParameterSet.bBusy THEN
			stMcAxisOnline.mcReadParameterSet.bExecute	:=	 FALSE;
			IF stMcAxisOnline.mcReadParameterSet.bDone THEN
				iInitStep 				:= iInitStep + 10;
				bReadParameterSetReady 	:= TRUE;
			ELSE
				iInitStep 				:= 1000;		// Error step
			END_IF
		END_IF	
	
	40:	// Get Drive Ref
		
		stMcAxisOnline.stGetDriveRef.bExecute		:=	 TRUE;
		iInitStep						:= iInitStep + 10;
		
	50: // Wait for data
	
		IF NOT stMcAxisOnline.stGetDriveRef.bBusy THEN
			stMcAxisOnline.stGetDriveRef.bExecute	:=	 FALSE;
			IF NOT stMcAxisOnline.stGetDriveRef.bError THEN
				iInitStep 				:= iInitStep + 10;
				bDriveRefReady 			:= TRUE;
			ELSE
				iInitStep 				:= 1000;		// Error step
			END_IF
		END_IF
	
	60: // Success - initialized flag, clear error
		bReInitialized					:= bInitialized;	// TRUE only when it's not first initialization e.g. online change
		bInitialized 					:= TRUE;
		bReInitializationError			:= FALSE;			// TRUE only when it's not first initialization e.g. online change
		bInitializationError			:= FALSE;
		iInitStep 						:= iInitStep + 10;
		
	70: // Idle
	
		;
		
	1000: // Error step
		wInitializationErrorCounter 	:= wInitializationErrorCounter + 1;
		IF wInitializationErrorCounter < 100 THEN
			iInitStep					:= iInitStep + 5;			// Go to delay
		ELSE
			bReInitializationError		:= bInitializationError;	// TRUE only when it's not first initialization e.g. online change
			bInitializationError		:= TRUE;
			bReInitialized				:= FALSE;
			iInitStep 					:= iInitStep + 10;
		END_IF

	1005: // Delay step
		tonDelay(IN:= TRUE, PT:= T#1S);
		IF tonDelay.Q THEN
			tonDelay(IN:= FALSE, PT:= T#1S);
			iInitStep					:= 0;
		END_IF
		
	1010: // Idle after error
		;
	
END_CASE

mcReadDriveAddress(	Axis				:= Axis,
					Execute				:= stMcAxisOnline.mcReadDriveAddress.bExecute,
					Done				=> stMcAxisOnline.mcReadDriveAddress.bDone,
					Busy				=> stMcAxisOnline.mcReadDriveAddress.bBusy,
					Error				=> stMcAxisOnline.mcReadDriveAddress.bError,
					ErrorID				=> stMcAxisOnline.mcReadDriveAddress.udiErrorID,
					DriveAddress		=> stMcAxisOnline.stDriveAddress);
				
mcReadParameterSet(	Parameter			:= stMcAxisOnline.stAxisParameter,
					Axis				:= Axis,
					Execute				:= stMcAxisOnline.mcReadParameterSet.bExecute,
					Done				=> stMcAxisOnline.mcReadParameterSet.bDone,
					Busy				=> stMcAxisOnline.mcReadParameterSet.bBusy,
					Error				=> stMcAxisOnline.mcReadParameterSet.bError,
					ErrorID				=> stMcAxisOnline.mcReadParameterSet.udiErrorID);
					
fbGetDriveRef(		bExecute			:= stMcAxisOnline.stGetDriveRef.bExecute,
					bBusy				=> stMcAxisOnline.stGetDriveRef.bBusy,
					bError				=> stMcAxisOnline.stGetDriveRef.bError,
					udiErrorID			=> stMcAxisOnline.stGetDriveRef.udiErrorID,
					stDriveRef			=> stMcAxisOnline.stDriveRef,
					Axis				:= Axis);
END_ACTION

ACTION ACT_Jog:
// Direct access from bSlow or bFast, if none then free choice
IF stMcAxisOnline.mcJog.bSlowForward OR stMcAxisOnline.mcJog.bSlowBackward THEN
	stMcAxisOnline.mcJog.eMode			:= MC_JOGMODE_STANDARD_SLOW;
ELSIF stMcAxisOnline.mcJog.bFastForward OR stMcAxisOnline.mcJog.bFastBackward THEN
	stMcAxisOnline.mcJog.eMode			:= MC_JOGMODE_STANDARD_FAST;
END_IF

mcJog(		Axis						:= Axis,
			JogForward					:= stMcAxisOnline.mcJog.bJogForward OR stMcAxisOnline.mcJog.bSlowForward OR stMcAxisOnline.mcJog.bFastForward,
			JogBackwards				:= stMcAxisOnline.mcJog.bJogBackwards OR stMcAxisOnline.mcJog.bSlowBackward OR stMcAxisOnline.mcJog.bFastBackward,
			Mode						:= stMcAxisOnline.mcJog.eMode,
			Position					:= stMcAxisOnline.mcJog.lrPosition,
			Velocity					:= stMcAxisOnline.mcJog.lrVelocity,
			Acceleration				:= stMcAxisOnline.mcJog.lrAcceleration,
			Deceleration				:= stMcAxisOnline.mcJog.lrDeceleration,
			Jerk						:= stMcAxisOnline.mcJog.lrJerk,
			Done						=> stMcAxisOnline.mcJog.bDone,
			Busy						=> stMcAxisOnline.mcJog.bBusy,
			Active						=> stMcAxisOnline.mcJog.bActive,
			CommandAborted				=> stMcAxisOnline.mcJog.bCommandAborted,
			Error						=> stMcAxisOnline.mcJog.bError,
			ErrorID						=> stMcAxisOnline.mcJog.udiErrorID);
END_ACTION

ACTION ACT_MotorMonitoring:
fbMotorMonitoring(
					bReset				:= stMcAxisOnline.stMotorMonitoring.bReset, 
					rTorqueLimit		:= stMcAxisOnline.stMotorMonitoring.rTorqueLimit , 
					bError				=> stMcAxisOnline.stMotorMonitoring.bError , 
					uiAdsErrId			=> stMcAxisOnline.stMotorMonitoring.uiAdsErrId , 
					uiSercosErrId		=> stMcAxisOnline.stMotorMonitoring.uiSecErrId, 
					bInitialized		=> stMcAxisOnline.stMotorMonitoring.bInitialized , 
					bWarning			=> stMcAxisOnline.stMotorMonitoring.bWarning , 
					rWarningCurrent		=> stMcAxisOnline.stMotorMonitoring.rWarningCurrent , 
					rTorquePerc			=> stMcAxisOnline.stMotorMonitoring.rTorquePerc,
					rTorquePercMax		=> stMcAxisOnline.stMotorMonitoring.rTorquePercMax,
					rTorque				=> stMcAxisOnline.stMotorMonitoring.rTorque , 
					rTorqueF			=> stMcAxisOnline.stMotorMonitoring.rTorqueF , 
					rTorqueMax			=> stMcAxisOnline.stMotorMonitoring.rTorqueMax , 
					rCurrent			=> stMcAxisOnline.stMotorMonitoring.rCurrent , 
					rCurrentF			=> stMcAxisOnline.stMotorMonitoring.rCurrentF , 
					rCurrentMax			=> stMcAxisOnline.stMotorMonitoring.rCurrentMax , 
					rI2T				=> stMcAxisOnline.stMotorMonitoring.rI2T , 
					rI2TMax				=> stMcAxisOnline.stMotorMonitoring.rI2TMax , 
					Axis				:= Axis );
END_ACTION

ACTION ACT_Move:
{region "Primary"}
mcMoveAbsolute(	Axis					:= Axis,
				Execute					:= stMcAxisOnline.mcMoveAbsolute.bExecute,
				Position				:= stMcAxisOnline.mcMoveAbsolute.lrPosition,
				Velocity				:= stMcAxisOnline.mcMoveAbsolute.lrVelocity,
				Acceleration			:= stMcAxisOnline.mcMoveAbsolute.lrAcceleration,
				Deceleration			:= stMcAxisOnline.mcMoveAbsolute.lrDeceleration,
				Jerk					:= stMcAxisOnline.mcMoveAbsolute.lrJerk,
				BufferMode				:= stMcAxisOnline.mcMoveAbsolute.eBufferMode,
				Options					:= stMcAxisOnline.mcMoveAbsolute.stOptions,
				Done					=> stMcAxisOnline.mcMoveAbsolute.bDone,
				Busy					=> stMcAxisOnline.mcMoveAbsolute.bBusy,
				Active					=> stMcAxisOnline.mcMoveAbsolute.bActive,
				CommandAborted			=> stMcAxisOnline.mcMoveAbsolute.bCommandAborted,
				Error					=> stMcAxisOnline.mcMoveAbsolute.bError,
				ErrorID					=> stMcAxisOnline.mcMoveAbsolute.udiErrorID);

mcMoveRelative(	Axis					:= Axis,
				Execute					:= stMcAxisOnline.mcMoveRelative.bExecute,
				Distance				:= stMcAxisOnline.mcMoveRelative.lrDistance,
				Velocity				:= stMcAxisOnline.mcMoveRelative.lrVelocity,
				Acceleration			:= stMcAxisOnline.mcMoveRelative.lrAcceleration,
				Deceleration			:= stMcAxisOnline.mcMoveRelative.lrDeceleration,
				Jerk					:= stMcAxisOnline.mcMoveRelative.lrJerk,
				BufferMode				:= stMcAxisOnline.mcMoveRelative.eBufferMode,
				Options					:= stMcAxisOnline.mcMoveRelative.stOptions,
				Done					=> stMcAxisOnline.mcMoveRelative.bDone,
				Busy					=> stMcAxisOnline.mcMoveRelative.bBusy,
				Active					=> stMcAxisOnline.mcMoveRelative.bActive,
				CommandAborted			=> stMcAxisOnline.mcMoveRelative.bCommandAborted,
				Error					=> stMcAxisOnline.mcMoveRelative.bError,
				ErrorID					=> stMcAxisOnline.mcMoveRelative.udiErrorID);
				
mcMoveVelocity(	Axis					:= Axis,
				Execute					:= stMcAxisOnline.mcMoveVelocity.bExecute,
				Velocity				:= stMcAxisOnline.mcMoveVelocity.lrVelocity,
				Acceleration			:= stMcAxisOnline.mcMoveVelocity.lrAcceleration,
				Deceleration			:= stMcAxisOnline.mcMoveVelocity.lrDeceleration,
				Jerk					:= stMcAxisOnline.mcMoveVelocity.lrJerk,
				Direction				:= stMcAxisOnline.mcMoveVelocity.eDirection,
				BufferMode				:= stMcAxisOnline.mcMoveVelocity.eBufferMode,
				Options					:= stMcAxisOnline.mcMoveVelocity.stOptions,
				InVelocity				=> stMcAxisOnline.mcMoveVelocity.bInVelocity,
				Busy					=> stMcAxisOnline.mcMoveVelocity.bBusy,
				Active					=> stMcAxisOnline.mcMoveVelocity.bActive,
				CommandAborted			=> stMcAxisOnline.mcMoveVelocity.bCommandAborted,
				Error					=> stMcAxisOnline.mcMoveVelocity.bError,
				ErrorID					=> stMcAxisOnline.mcMoveVelocity.udiErrorID);
stMcAxisOnline.mcMoveVelocity.bDone		:= stMcAxisOnline.mcMoveVelocity.bInVelocity;

mcMoveModulo(	Axis					:= Axis,
				Execute					:= stMcAxisOnline.mcMoveModulo.bExecute,
				Position				:= stMcAxisOnline.mcMoveModulo.lrPosition,
				Velocity				:= stMcAxisOnline.mcMoveModulo.lrVelocity,
				Acceleration			:= stMcAxisOnline.mcMoveModulo.lrAcceleration,
				Deceleration			:= stMcAxisOnline.mcMoveModulo.lrDeceleration,
				Jerk					:= stMcAxisOnline.mcMoveModulo.lrJerk,
				Direction				:= stMcAxisOnline.mcMoveModulo.eDirection,
				BufferMode				:= stMcAxisOnline.mcMoveModulo.eBufferMode,
				Options					:= stMcAxisOnline.mcMoveModulo.stOptions,
				Done					=> stMcAxisOnline.mcMoveModulo.bDone,
				Busy					=> stMcAxisOnline.mcMoveModulo.bBusy,
				Active					=> stMcAxisOnline.mcMoveModulo.bActive,
				CommandAborted			=> stMcAxisOnline.mcMoveModulo.bCommandAborted,
				Error					=> stMcAxisOnline.mcMoveModulo.bError,
				ErrorID					=> stMcAxisOnline.mcMoveModulo.udiErrorID);
{endregion}
{region "Secondary"}
mcMoveAbsolute2(Axis					:= Axis,
				Execute					:= stMcAxisOnline.mcMoveAbsolute2.bExecute,
				Position				:= stMcAxisOnline.mcMoveAbsolute2.lrPosition,
				Velocity				:= stMcAxisOnline.mcMoveAbsolute2.lrVelocity,
				Acceleration			:= stMcAxisOnline.mcMoveAbsolute2.lrAcceleration,
				Deceleration			:= stMcAxisOnline.mcMoveAbsolute2.lrDeceleration,
				Jerk					:= stMcAxisOnline.mcMoveAbsolute2.lrJerk,
				BufferMode				:= stMcAxisOnline.mcMoveAbsolute2.eBufferMode,
				Options					:= stMcAxisOnline.mcMoveAbsolute2.stOptions,
				Done					=> stMcAxisOnline.mcMoveAbsolute2.bDone,
				Busy					=> stMcAxisOnline.mcMoveAbsolute2.bBusy,
				Active					=> stMcAxisOnline.mcMoveAbsolute2.bActive,
				CommandAborted			=> stMcAxisOnline.mcMoveAbsolute2.bCommandAborted,
				Error					=> stMcAxisOnline.mcMoveAbsolute2.bError,
				ErrorID					=> stMcAxisOnline.mcMoveAbsolute2.udiErrorID);

mcMoveRelative2(Axis					:= Axis,
				Execute					:= stMcAxisOnline.mcMoveRelative2.bExecute,
				Distance				:= stMcAxisOnline.mcMoveRelative2.lrDistance,
				Velocity				:= stMcAxisOnline.mcMoveRelative2.lrVelocity,
				Acceleration			:= stMcAxisOnline.mcMoveRelative2.lrAcceleration,
				Deceleration			:= stMcAxisOnline.mcMoveRelative2.lrDeceleration,
				Jerk					:= stMcAxisOnline.mcMoveRelative2.lrJerk,
				BufferMode				:= stMcAxisOnline.mcMoveRelative2.eBufferMode,
				Options					:= stMcAxisOnline.mcMoveRelative2.stOptions,
				Done					=> stMcAxisOnline.mcMoveRelative2.bDone,
				Busy					=> stMcAxisOnline.mcMoveRelative2.bBusy,
				Active					=> stMcAxisOnline.mcMoveRelative2.bActive,
				CommandAborted			=> stMcAxisOnline.mcMoveRelative2.bCommandAborted,
				Error					=> stMcAxisOnline.mcMoveRelative2.bError,
				ErrorID					=> stMcAxisOnline.mcMoveRelative2.udiErrorID);
				
mcMoveVelocity2(Axis					:= Axis,
				Execute					:= stMcAxisOnline.mcMoveVelocity2.bExecute,
				Velocity				:= stMcAxisOnline.mcMoveVelocity2.lrVelocity,
				Acceleration			:= stMcAxisOnline.mcMoveVelocity2.lrAcceleration,
				Deceleration			:= stMcAxisOnline.mcMoveVelocity2.lrDeceleration,
				Jerk					:= stMcAxisOnline.mcMoveVelocity2.lrJerk,
				Direction				:= stMcAxisOnline.mcMoveVelocity2.eDirection,
				BufferMode				:= stMcAxisOnline.mcMoveVelocity2.eBufferMode,
				Options					:= stMcAxisOnline.mcMoveVelocity2.stOptions,
				InVelocity				=> stMcAxisOnline.mcMoveVelocity2.bInVelocity,
				Busy					=> stMcAxisOnline.mcMoveVelocity2.bBusy,
				Active					=> stMcAxisOnline.mcMoveVelocity2.bActive,
				CommandAborted			=> stMcAxisOnline.mcMoveVelocity2.bCommandAborted,
				Error					=> stMcAxisOnline.mcMoveVelocity2.bError,
				ErrorID					=> stMcAxisOnline.mcMoveVelocity2.udiErrorID);
stMcAxisOnline.mcMoveVelocity2.bDone	:= stMcAxisOnline.mcMoveVelocity2.bInVelocity;

mcMoveModulo2(	Axis					:= Axis,
				Execute					:= stMcAxisOnline.mcMoveModulo2.bExecute,
				Position				:= stMcAxisOnline.mcMoveModulo2.lrPosition,
				Velocity				:= stMcAxisOnline.mcMoveModulo2.lrVelocity,
				Acceleration			:= stMcAxisOnline.mcMoveModulo2.lrAcceleration,
				Deceleration			:= stMcAxisOnline.mcMoveModulo2.lrDeceleration,
				Jerk					:= stMcAxisOnline.mcMoveModulo2.lrJerk,
				Direction				:= stMcAxisOnline.mcMoveModulo2.eDirection,
				BufferMode				:= stMcAxisOnline.mcMoveModulo2.eBufferMode,
				Options					:= stMcAxisOnline.mcMoveModulo2.stOptions,
				Done					=> stMcAxisOnline.mcMoveModulo2.bDone,
				Busy					=> stMcAxisOnline.mcMoveModulo2.bBusy,
				Active					=> stMcAxisOnline.mcMoveModulo2.bActive,
				CommandAborted			=> stMcAxisOnline.mcMoveModulo2.bCommandAborted,
				Error					=> stMcAxisOnline.mcMoveModulo2.bError,
				ErrorID					=> stMcAxisOnline.mcMoveModulo2.udiErrorID);
{endregion}
END_ACTION

ACTION ACT_Power:
mcPower(	Axis						:= Axis,									//
			Enable						:= stMcAxisOnline.mcPower.bEnable,
			Enable_Positive				:= stMcAxisOnline.mcPower.bEnable_Positive,
			Enable_Negative				:= stMcAxisOnline.mcPower.bEnable_Negative,
			Override					:= stMcAxisOnline.mcPower.lrOverride,
			BufferMode					:= stMcAxisOnline.mcPower.eBufferMode,
			Options						:= stMcAxisOnline.mcPower.stOptions,
			Status						=> stMcAxisOnline.mcPower.bStatus,
			Busy						=> stMcAxisOnline.mcPower.bBusy,
			Active						=> stMcAxisOnline.mcPower.bActive,
			Error						=> stMcAxisOnline.mcPower.bError,
			ErrorID						=> stMcAxisOnline.mcPower.udiErrorID);
END_ACTION

ACTION ACT_ResetAndDiag:
tonGetDriveDiag(IN:= stMcAxisOnline.stError.bDriveError AND NOT tonGetDriveDiag.Q, PT:= T#5S, Q=> , ET=> );

IF Axis.Status.OpMode.SimulationAxis THEN
	mcReset(
		Axis						:= Axis,
		Execute						:= stMcAxisOnline.mcReset.bExecute,
		Done						=> stMcAxisOnline.mcReset.bDone,
		Busy						=> stMcAxisOnline.mcReset.bBusy,
		Error						=> stMcAxisOnline.mcReset.bError,
		ErrorID						=> stMcAxisOnline.mcReset.udiErrorID);	
ELSE
	fbReadChannelErrorCode(
		Reset:=					stMcAxisOnline.mcReset.bExecute,
		GetDiag				:=	(stMcAxisOnline.stChannelErrorCode.bExecute OR tonGetDriveDiag.Q),
		Axis				:=	Axis , 
		stAX5000Diag		:=	stAX5000Diag , 
		Error				=> 	stMcAxisOnline.mcReset.bError , 
		AdsErrId			=>	stMcAxisOnline.mcReset.udiErrorID , 
		SercosErrId			=>	stMcAxisOnline.stChannelErrorCode.uiAdsErrId, //???
		ResetAct			=> , 
		DiagAct				=> , 
		Busy				=> 	stMcAxisOnline.mcReset.bBusy );
	
	stMcAxisOnline.stChannelErrorCode.bError 				:= stAX5000Diag.bC1DError;
	stMcAxisOnline.stChannelErrorCode.uiChannelErrorCode 	:= UDINT_TO_UINT (stAX5000Diag.iDiagNumber);
	stMcAxisOnline.stChannelErrorCode.uiChannelErrorCodeHex := UDINT_TO_UINT (stAX5000Diag.iDiagNumber);
END_IF
END_ACTION

ACTION ACT_SetPosition:
mcSetPosition(		Axis				:= Axis,
					Execute				:= stMcAxisOnline.mcSetPosition.bExecute,
					Position			:= stMcAxisOnline.mcSetPosition.lrPosition,
					Mode				:= stMcAxisOnline.mcSetPosition.bMode,
					Options				:= stMcAxisOnline.mcSetPosition.stOptions,
					Done				=> stMcAxisOnline.mcSetPosition.bDone,
					Busy				=> stMcAxisOnline.mcSetPosition.bBusy,
					Error				=> stMcAxisOnline.mcSetPosition.bError,
					ErrorID				=> stMcAxisOnline.mcSetPosition.udiErrorID);
END_ACTION

ACTION ACT_SetPositionIO:
fbSetPositionOffset(
	bExecute			:= stMcAxisOnline.stSetPositionOffset.bExecute , 
	lrPosition			:= stMcAxisOnline.stSetPositionOffset.lrPosition , 
	bRelative			:= stMcAxisOnline.stSetPositionOffset.bRelative , 
	eFeedback			:= stMcAxisOnline.stSetPositionOffset.eFeedback , 
	eMemory				:= stMcAxisOnline.stSetPositionOffset.eMemory , 
	bBusy				=> stMcAxisOnline.stSetPositionOffset.bBusy , 
	bError				=> stMcAxisOnline.stSetPositionOffset.bError, 
	udiErrorID			=> stMcAxisOnline.stSetPositionOffset.udiErrorID, 
	uiSoEErrorID		=> stMcAxisOnline.stSetPositionOffset.uiSecErrId,
	Axis				:= Axis );
END_ACTION

ACTION ACT_States:
// Read States and forward main states
Axis.ReadStatus();
stMcAxisOnline.stStatus.stAxisStatus		:= Axis.Status;
stMcAxisOnline.stStatus.dwAxisId			:= Axis.NcToPlc.AxisId;
stMcAxisOnline.stStatus.bNcError			:= Axis.Status.Error;
stMcAxisOnline.stStatus.udiNcErrorCode		:= Axis.Status.ErrorID;
stMcAxisOnline.stStatus.udiNcErrorCodeHex	:= Axis.Status.ErrorID;

stMcAxisOnline.stStatus.sAxisName			:= stMcAxisOnline.stAxisParameter.sAxisName;
stMcAxisOnline.stStatus.lrActPos			:= Axis.NcToPlc.ActPos;
stMcAxisOnline.stStatus.lrModuloActPos		:= Axis.NcToPlc.ModuloActPos;
stMcAxisOnline.stStatus.lrActVelo			:= Axis.NcToPlc.ActVelo;
stMcAxisOnline.stStatus.lrActAcc			:= Axis.NcToPlc.ActAcc;
stMcAxisOnline.stStatus.lrActTorque			:= Axis.NcToPlc.ActTorque;
stMcAxisOnline.stStatus.lrPosDiff			:= Axis.NcToPlc.PosDiff;
stMcAxisOnline.stStatus.lrSetPos			:= Axis.NcToPlc.SetPos;
stMcAxisOnline.stStatus.lrSetVelo			:= Axis.NcToPlc.SetVelo;
stMcAxisOnline.stStatus.lrSetAcc			:= Axis.NcToPlc.SetAcc;
stMcAxisOnline.stStatus.lrSetTorque			:= Axis.NcToPlc.SetTorque;
stMcAxisOnline.stStatus.lrPosDiff			:= Axis.NcToPlc.PosDiff;
stMcAxisOnline.stStatus.bAxisReady			:= Axis.Status.Operational;
stMcAxisOnline.stStatus.bHomed				:= Axis.Status.Homed;
stMcAxisOnline.stStatus.bCoupled			:= Axis.Status.Coupled;

// zezwolenie na zjazd z krancowki hw
Axis.PlcToNc.ControlDWord.8				:= stMcAxisOnline.stStatus.bAcceptBlockedDrive;
END_ACTION

ACTION ACT_Stop:
mcHalt(		Axis						:= Axis,
			Execute						:= stMcAxisOnline.mcHalt.bExecute,
			Deceleration				:= stMcAxisOnline.mcHalt.lrDeceleration,
			Jerk						:= stMcAxisOnline.mcHalt.lrJerk,
			BufferMode					:= stMcAxisOnline.mcHalt.eBufferMode,
			Options						:= stMcAxisOnline.mcHalt.stOptions,
			Done						=> stMcAxisOnline.mcHalt.bDone,
			Busy						=> stMcAxisOnline.mcHalt.bBusy,
			Active						=> stMcAxisOnline.mcHalt.bActive,
			CommandAborted				=> stMcAxisOnline.mcHalt.bCommandAborted,
			Error						=> stMcAxisOnline.mcHalt.bError,
			ErrorID						=> stMcAxisOnline.mcHalt.udiErrorID);
			
mcStop(		Axis						:= Axis,
			Execute						:= stMcAxisOnline.mcStop.bExecute,
			Deceleration				:= stMcAxisOnline.mcStop.lrDeceleration,
			Jerk						:= stMcAxisOnline.mcStop.lrJerk,
			Options						:= stMcAxisOnline.mcStop.stOptions,
			Done						=> stMcAxisOnline.mcStop.bDone,
			Busy						=> stMcAxisOnline.mcStop.bBusy,
			Active						=> stMcAxisOnline.mcStop.bActive,
			CommandAborted				=> stMcAxisOnline.mcStop.bCommandAborted,
			Error						=> stMcAxisOnline.mcStop.bError,
			ErrorID						=> stMcAxisOnline.mcStop.udiErrorID);
			
mcStopSS2(	Axis						:= Axis,
			Execute						:= stMcAxisOnline.mcSS2.bExecute,
			Deceleration				:= stMcAxisOnline.mcSS2.lrDeceleration,
			Jerk						:= stMcAxisOnline.mcSS2.lrJerk,
			Options						:= stMcAxisOnline.mcSS2.stOptions,
			Done						=> stMcAxisOnline.mcSS2.bDone,
			Busy						=> stMcAxisOnline.mcSS2.bBusy,
			Active						=> stMcAxisOnline.mcSS2.bActive,
			CommandAborted				=> stMcAxisOnline.mcSS2.bCommandAborted,
			Error						=> stMcAxisOnline.mcSS2.bError,
			ErrorID						=> stMcAxisOnline.mcSS2.udiErrorID);
			
mcStopSS1(	Axis						:= Axis,
			Execute						:= stMcAxisOnline.mcSS1.bExecute,
			Deceleration				:= stMcAxisOnline.mcSS1.lrDeceleration,
			Jerk						:= stMcAxisOnline.mcSS1.lrJerk,
			Options						:= stMcAxisOnline.mcSS1.stOptions,
			Done						=> stMcAxisOnline.mcSS1.bDone,
			Busy						=> stMcAxisOnline.mcSS1.bBusy,
			Active						=> stMcAxisOnline.mcSS1.bActive,
			CommandAborted				=> stMcAxisOnline.mcSS1.bCommandAborted,
			Error						=> stMcAxisOnline.mcSS1.bError,
			ErrorID						=> stMcAxisOnline.mcSS1.udiErrorID);
// SS1 - after MC_Stop function we have to disable drive			
stMcAxisOnline.mcPower.bEnable R= stMcAxisOnline.mcPower.bEnable_Positive R= stMcAxisOnline.mcPower.bEnable_Negative R= (stMcAxisOnline.mcSS1.bDone OR stMcAxisOnline.mcSS1.bCommandAborted OR stMcAxisOnline.mcSS1.bError);
END_ACTION

ACTION ACT_SWLimitSwitch:
fbNcLimitSwitch(	udiAxisID		:= Axis.NcToPlc.AxisId, 
					bRead			:= stMcAxisOnline.stNcLimitSwitch.bRead, 
					bWrite			:= stMcAxisOnline.stNcLimitSwitch.bWrite, 
					bReset			:= stMcAxisOnline.stNcLimitSwitch.bReset, 
					lrSetMinPos		:= stMcAxisOnline.stNcLimitSwitch.lrSetMinPos, 
					lrSetMaxPos		:= stMcAxisOnline.stNcLimitSwitch.lrSetMaxPos, 
					bSetMinMon		:= stMcAxisOnline.stNcLimitSwitch.bSetMinMon, 
					bSetMaxMon		:= stMcAxisOnline.stNcLimitSwitch.bSetMaxMon, 
					bBusy			=> stMcAxisOnline.stNcLimitSwitch.bBusy, 
					bError			=> stMcAxisOnline.stNcLimitSwitch.bError, 
					udiErrorID		=> stMcAxisOnline.stNcLimitSwitch.udiErrorID, 
					lrActMinPos		=> stMcAxisOnline.stNcLimitSwitch.lrActMinPos, 
					lrActMaxPos		=> stMcAxisOnline.stNcLimitSwitch.lrActMaxPos, 
					bActMinMon		=> stMcAxisOnline.stNcLimitSwitch.bActMinMon, 
					bActMaxMon		=> stMcAxisOnline.stNcLimitSwitch.bActMaxMon);
END_ACTION

END_FUNCTION_BLOCK

// ---- POUs/POUsAxisOnline/AX5000/FB_SetPositionOffset.TcPOU
//==================================================================================================
//							Beckhoff Automation Poland
//									07.06.2018
//	Blok do uzupełniania offsetu w enkoderze/AX5000
//	Obsluguje bledy zwiazane z wymiana silnika na nowy - bez wpisanego offsetu.
//	Naprawia błąd: 	0x0000F340- Position offset invalid.
//					0x0000F341- Position offset: No position offset excisting.
//	Aby wpisać wartość, silnik musi być wyłączony.
//	Niezbędne biblioteki:
//	Tc2_MC2;	Tc2_Utilities;	Tc2_MC2_Drive;	Tc2_EtherCAT, Tc2_Drive;
//
//	v2.4 || TC v 3.1.4022.20 || - Usuniecie nieużywanych zmiennych, zabezpieczenie przed zerowa pozycja, optymalizacje
//	v2.2 || TC v 3.1.4022.2	 || - Poprawka w komentarzu, uiSoEErrorID zamiast udiSoEErrorID
//	v2.1 || TC v 3.1.4022.0	 || - Uproszczono kod
//	v2.0 || TC v 3.1.4022.0	 || - Dodano obsługę AX52xx, przebudowano bloczek z wykorzystaniem FB_ChangeSlaveState
//	v1.0 || TC v 3.1.4020.32 || - Pierwsza wersja
//==================================================================================================
FUNCTION_BLOCK FB_SetPositionOffset
VAR_INPUT
	bExecute								: BOOL;							// rising edge starts sequence
	lrPosition								: LREAL		:=	0.001;			// Write new encoder position
	bRelative								: BOOL;							// When this flag is set, the position is relatively interpreted
	eFeedback								: E_PositionOffsetFeedback;		// ePositionOffsetFeedback1:= 0			ePositionOffsetFeedback2 := 1
	eMemory									: E_PositionOffsetMemory;		// ePositionOffsetMemory_Encoder:= 0	ePositionOffsetMemory_Drive := 1
END_VAR
VAR_OUTPUT
	bBusy									: BOOL;
	bError									: BOOL;	
	udiErrorID								: UDINT;						// bError=TRUE AND udiErrorID=0 means state request timeout
	uiSoEErrorID							: UINT;
	udiADSerrorID							: UDINT;
END_VAR
VAR_IN_OUT
	Axis									: AXIS_REF;
END_VAR
VAR CONSTANT
	NCIDXG_AXPARMS							: UDINT			:= 16#4000;		// ADS group number to axis parameters 
	NCIDXO_AXP_HWAMSADDR					: UDINT			:= 16#31;		// ADS offset to drive channel
END_VAR
VAR
	rtExecute								: R_TRIG;						// bExecute triggers start
	fbSoEReset								: FB_SoEReset;
	fbSoEWritePassword						: FB_SoEWritePassword;			// unlock P-0-0278
	fbSoEAX5000SetPositionOffset			: FB_SoEAX5000SetPositionOffset;
	fbSoEReadDiagNumber						: FB_SoEReadDiagNumber;	
	fbSoEWrite_ByDriveRef					: FB_SoEWrite_ByDriveRef;
	fbSoERead_ByDriveRef					: FB_SoERead_ByDriveRef;
	fbChangeSlaveState						: FB_ChangeEtherCATSlaveState;
	fbAdsRead								: ADSREAD;
	stPlcDriveRef							: ST_PlcDriveRef;				// ADS buffer (need to change aNetId into sNetId)
	stDriveRef								: ST_DriveRef;					// come from stPlcDriveRef
	bDualChannel							: BOOL;
	stSoE_String							: ST_SoE_String;				// buffer for byDualChannel
	P_0_0278_Value							: WORD;							//	0- NO	1- YES
	iStep									: INT;							// Actual Step
	iLastStep								: INT;							// Last step before error
END_VAR

rtExecute	(CLK:= bExecute );

CASE iStep	OF

	0:																//	Enable FB, lock input parameters
		IF rtExecute.Q THEN
			bBusy							:= TRUE;
			bError							:= FALSE;
			udiErrorID						:= 0;
			uiSoEErrorID					:= 0;
			udiADSerrorID					:= 0;
			iLastStep						:= 0;
			IF ABS(lrPosition) < LREAL#0.0001 THEN
				fbSoEAX5000SetPositionOffset.Position := LREAL#0.0001;
			ELSE
				fbSoEAX5000SetPositionOffset.Position := lrPosition; 
			END_IF
			fbSoEAX5000SetPositionOffset.Memory	:= eMemory;
			fbSoEAX5000SetPositionOffset.Relative := bRelative;
			fbSoEAX5000SetPositionOffset.Feedback := eFeedback;
			iStep							:= iStep+10;
		END_IF			

	10:																// Get Drive channel from AXIS_REF by ADS
		fbAdsRead.NETID						:= '';
		fbAdsRead.PORT						:= AMSPORT_R0_NC;		// set ADS Port to NC
		fbAdsRead.IDXGRP					:= NCIDXG_AXPARMS + Axis.NcToPlc.AxisId;	// set ADS Group to AXIS Parameters
		fbAdsRead.IDXOFFS					:= NCIDXO_AXP_HWAMSADDR;// set ADS offset to channel number
		fbAdsRead.LEN						:= SIZEOF(stPlcDriveRef);
		fbAdsRead.DESTADDR					:= ADR(stPlcDriveRef);
		fbAdsRead.TMOUT						:= T#5S;
		fbAdsRead.READ						:= TRUE;
		iStep								:= istep+10;
		
	20:																// reading actual channel (DriveNo) from AXIS_REF	
		fbAdsRead.READ						:= FALSE;
		IF NOT fbAdsRead.BUSY THEN
			IF  NOT fbAdsRead.ERR THEN
				iStep							:= iStep+10;	
				stDriveRef.sNetId				:= F_CreateAmsNetId(stPlcDriveRef.aNetId);	// change AmsNetId array into string
				stDriveRef.nSlaveAddr			:= stPlcDriveRef.nSlaveAddr;
				stDriveRef.nDriveNo				:= stPlcDriveRef.nDriveNo;	
				fbChangeSlaveState.sEtherCAT_NetID:= stDriveRef.sNetId;
				fbChangeSlaveState.nSlaveAddr	:= stDriveRef.nSlaveAddr;
			ELSIF fbAdsRead.ERR THEN
				udiADSerrorID					:= fbAdsRead.ERRID;
				iLastStep						:= iStep;
				iStep							:= 999;				
			END_IF
		END_IF
		
	30:																// Read drive diag number
		fbSoEReadDiagNumber.NetId			:= '';
		fbSoEReadDiagNumber.Execute			:= TRUE;
		iStep								:= iStep+10;

	40:																// Choose method
		fbSoEReadDiagNumber.Execute			:= FALSE;
		IF NOT fbSoEReadDiagNumber.Busy THEN
			IF fbSoEReadDiagNumber.DiagNumber = (16#F341 OR 16#F340) THEN
				iStep						:= 50;					// Position errors -> Reset errors and write 
			ELSIF	fbSoEReadDiagNumber.DiagNumber >= (16#F000) THEN
				iLastStep					:= iStep;				// Do nothing in other error states
				iStep						:= 999;
			ELSE												
				iStep						:= 200;					// Drive Ready -> Write without changing OP State			
			END_IF
		END_IF
	
	50:																// Request INIT State
		fbChangeSlaveState.byReguestedState	:= EC_DEVICE_STATE_INIT;
		fbChangeSlaveState.bExecute			:= TRUE;
		iStep								:= iStep+10;

	60,80:															// Wait till state changed
		fbChangeSlaveState.bExecute			:= FALSE;
		IF NOT fbChangeSlaveState.bBusy THEN
			IF NOT fbChangeSlaveState.bError THEN
				iStep							:= iStep+10;
			ELSE
				udiErrorID						:= fbChangeSlaveState.udiErrorID;
				iLastStep						:= iStep;
				iStep 							:= 999;
			END_IF
		END_IF
		
	70:																// Request PreOP State	
		fbChangeSlaveState.byReguestedState	:= EC_DEVICE_STATE_PREOP;
		fbChangeSlaveState.bExecute			:= TRUE;
		iStep								:= iStep+10;
		
	90:																// Write drive password (unlock P-0-0278)
		fbSoEWritePassword.Password.strData	:= 'AX5000';
		fbSoEWritePassword.NetId			:= '';
		fbSoEWritePassword.Execute			:= TRUE;
		iStep								:= iStep + 10;
		
